LIN {X 0,Y 362.001,Z 141.011,A -85,B 0,C 180,E1 -12973.899,E2 -12973.899} C_VEL
LIN {X 0,Y 361.93,Z 141.028,A -85,B 0,C 180,E1 -12976.934,E2 -12976.934} C_VEL
LIN {X 0,Y 361.889,Z 141.033,A -85,B 0,C 180,E1 -12980.461,E2 -12980.461} C_VEL
LIN {X 0,Y 361.895,Z 141.031,A -85,B 0,C 180,E1 -12984.112,E2 -12984.112} C_VEL
LIN {X 0,Y 361.866,Z 141.033,A -85,B 0,C 180,E1 -12987.782,E2 -12987.782} C_VEL
LIN {X 0,Y 361.849,Z 141.037,A -85,B 0,C 180,E1 -12991.285,E2 -12991.285} C_VEL
LIN {X 0,Y 361.856,Z 141.029,A -85,B 0,C 180,E1 -12994.28,E2 -12994.28} C_VEL
LIN {X 0,Y 361.864,Z 141.03,A -85,B 0,C 180,E1 -12997.223,E2 -12997.223} C_VEL
LIN {X 0,Y 361.836,Z 141.038,A -85,B 0,C 180,E1 -13000.755,E2 -13000.755} C_VEL
LIN {X 0,Y 361.818,Z 141.04,A -85,B 0,C 180,E1 -13004.368,E2 -13004.368} C_VEL
LIN {X 0,Y 361.837,Z 141.036,A -85,B 0,C 180,E1 -13007.568,E2 -13007.568} C_VEL
LIN {X 0,Y 361.871,Z 141.028,A -85,B 0,C 180,E1 -13010.973,E2 -13010.973} C_VEL
LIN {X 0,Y 361.89,Z 141.148,A -85,B 0,C 180,E1 -13012.93,E2 -13012.93} C_VEL
LIN {X 0,Y 365.148,Z 152.964,A -85,B 0,C 180,E1 -13015.855,E2 -13015.855} C_VEL
LIN {X 0,Y 367.944,Z 164.217,A -85,B 0,C 180,E1 -13018.43,E2 -13018.43} C_VEL
LIN {X 0,Y 374.959,Z 180.061,A -85,B 0,C 180,E1 -13019.427,E2 -13019.427} C_VEL
LIN {X 0,Y 380.015,Z 206.73,A -85,B 0,C 180,E1 -13020.441,E2 -13020.441} C_VEL
LIN {X 0,Y 378.027,Z 291.914,A -85,B 0,C 180,E1 -13022.078,E2 -13022.078} C_VEL
LIN {X 0,Y 376.936,Z 331.246,A -85,B 0,C 180,E1 -13022.856,E2 -13022.856} C_VEL
LIN {X 0,Y 375.915,Z 347.066,A -85,B 0,C 180,E1 -13023.377,E2 -13023.377} C_VEL
LIN {X 0,Y 374.628,Z 361.61,A -85,B 0,C 180,E1 -13024.065,E2 -13024.065} C_VEL
LIN {X 0,Y 373.287,Z 375.171,A -85,B 0,C 180,E1 -13024.921,E2 -13024.921} C_VEL
LIN {X 0,Y 371.559,Z 388.868,A -85,B 0,C 180,E1 -13026.004,E2 -13026.004} C_VEL
LIN {X 0,Y 369.85,Z 401.312,A -85,B 0,C 180,E1 -13027.221,E2 -13027.221} C_VEL
LIN {X 0,Y 367.894,Z 413.971,A -85,B 0,C 180,E1 -13028.718,E2 -13028.718} C_VEL
LIN {X 0,Y 366.21,Z 426.144,A -85,B 0,C 180,E1 -13030.483,E2 -13030.483} C_VEL
LIN {X 0,Y 364.434,Z 436.665,A -85,B 0,C 180,E1 -13032.318,E2 -13032.318} C_VEL
LIN {X 0,Y 363.094,Z 445.935,A -85,B 0,C 180,E1 -13034.277,E2 -13034.277} C_VEL
LIN {X 0,Y 361.936,Z 454.664,A -85,B 0,C 180,E1 -13036.525,E2 -13036.525} C_VEL
LIN {X 0,Y 361.134,Z 461.674,A -85,B 0,C 180,E1 -13038.778,E2 -13038.778} C_VEL
LIN {X 0,Y 360.628,Z 467.188,A -85,B 0,C 180,E1 -13041.031,E2 -13041.031} C_VEL
LIN {X 0,Y 360.386,Z 471.36,A -85,B 0,C 180,E1 -13043.28,E2 -13043.28} C_VEL
LIN {X 0,Y 360.3,Z 474.286,A -85,B 0,C 180,E1 -13045.525,E2 -13045.525} C_VEL
LIN {X 0,Y 360.254,Z 476.03,A -85,B 0,C 180,E1 -13047.764,E2 -13047.764} C_VEL
LIN {X 0,Y 360.357,Z 476.63,A -85,B 0,C 180,E1 -13050,E2 -13050} C_VEL
LIN {X 0,Y 360.254,Z 476.023,A -85,B 0,C 180,E1 -13052.236,E2 -13052.236} C_VEL
LIN {X 0,Y 360.302,Z 474.27,A -85,B 0,C 180,E1 -13054.475,E2 -13054.475} C_VEL
LIN {X 0,Y 360.387,Z 471.339,A -85,B 0,C 180,E1 -13056.719,E2 -13056.719} C_VEL
LIN {X 0,Y 360.628,Z 467.166,A -85,B 0,C 180,E1 -13058.969,E2 -13058.969} C_VEL
LIN {X 0,Y 361.126,Z 461.64,A -85,B 0,C 180,E1 -13061.222,E2 -13061.222} C_VEL
LIN {X 0,Y 361.911,Z 454.613,A -85,B 0,C 180,E1 -13063.476,E2 -13063.476} C_VEL
LIN {X 0,Y 363.094,Z 445.876,A -85,B 0,C 180,E1 -13065.723,E2 -13065.723} C_VEL
LIN {X 0,Y 364.405,Z 436.598,A -85,B 0,C 180,E1 -13067.683,E2 -13067.683} C_VEL
LIN {X 0,Y 366.146,Z 426.204,A -85,B 0,C 180,E1 -13069.497,E2 -13069.497} C_VEL
LIN {X 0,Y 367.737,Z 414.949,A -85,B 0,C 180,E1 -13071.145,E2 -13071.145} C_VEL
LIN {X 0,Y 369.626,Z 402.491,A -85,B 0,C 180,E1 -13072.646,E2 -13072.646} C_VEL
LIN {X 0,Y 371.34,Z 390.238,A -85,B 0,C 180,E1 -13073.863,E2 -13073.863} C_VEL
LIN {X 0,Y 373.143,Z 376.327,A -85,B 0,C 180,E1 -13074.981,E2 -13074.981} C_VEL
LIN {X 0,Y 374.607,Z 361.964,A -85,B 0,C 180,E1 -13075.898,E2 -13075.898} C_VEL
LIN {X 0,Y 375.898,Z 346.851,A -85,B 0,C 180,E1 -13076.62,E2 -13076.62} C_VEL
LIN {X 0,Y 376.854,Z 331.928,A -85,B 0,C 180,E1 -13077.113,E2 -13077.113} C_VEL
LIN {X 0,Y 377.84,Z 296.547,A -85,B 0,C 180,E1 -13077.824,E2 -13077.824} C_VEL
LIN {X 0,Y 380.046,Z 207.189,A -85,B 0,C 180,E1 -13079.53,E2 -13079.53} C_VEL
LIN {X 0,Y 375.356,Z 182.22,A -85,B 0,C 180,E1 -13080.473,E2 -13080.473} C_VEL
LIN {X 0,Y 374.41,Z 178.644,A -85,B 0,C 180,E1 -13080.636,E2 -13080.636} C_VEL
LIN {X 0,Y 367.8,Z 163.722,A -85,B 0,C 180,E1 -13081.611,E2 -13081.611} C_VEL
LIN {X 0,Y 364.582,Z 150.743,A -85,B 0,C 180,E1 -13084.657,E2 -13084.657} C_VEL
LIN {X 0,Y 361.877,Z 141.032,A -85,B 0,C 180,E1 -13087.125,E2 -13087.125} C_VEL
LIN {X 0,Y 361.836,Z 141.036,A -85,B 0,C 180,E1 -13090.756,E2 -13090.756} C_VEL
LIN {X 0,Y 361.818,Z 141.037,A -85,B 0,C 180,E1 -13094.369,E2 -13094.369} C_VEL
LIN {X 0,Y 361.837,Z 141.038,A -85,B 0,C 180,E1 -13097.568,E2 -13097.568} C_VEL
LIN {X 0,Y 361.869,Z 141.032,A -85,B 0,C 180,E1 -13100.974,E2 -13100.974} C_VEL
LIN {X 0,Y 361.875,Z 141.026,A -85,B 0,C 180,E1 -13104.655,E2 -13104.655} C_VEL
LIN {X 0,Y 361.838,Z 141.034,A -85,B 0,C 180,E1 -13108.371,E2 -13108.371} C_VEL
LIN {X 0,Y 361.902,Z 141.026,A -85,B 0,C 180,E1 -13110.955,E2 -13110.955} C_VEL
LIN {X 0,Y 361.955,Z 141.02,A -85,B 0,C 180,E1 -13113.475,E2 -13113.475} C_VEL
LIN {X 0,Y 361.88,Z 141.031,A -85,B 0,C 180,E1 -13117.144,E2 -13117.144} C_VEL
LIN {X 0,Y 361.907,Z 141.025,A -85,B 0,C 180,E1 -13120.724,E2 -13120.724} C_VEL
LIN {X 0,Y 361.934,Z 141.021,A -85,B 0,C 180,E1 -13123.066,E2 -13123.066} C_VEL
LIN {X 0,Y 362.001,Z 141.017,A -85,B 0,C 180,E1 -13126.528,E2 -13126.528} C_VEL
LIN {X 0,Y 362.002,Z 141.016,A -85,B 0,C 180,E1 -13129.937,E2 -13129.937} C_VEL
LIN {X 0,Y 362.126,Z 141.001,A -85,B 0,C 180,E1 -13133.313,E2 -13133.313} C_VEL
LIN {X 0,Y 362.279,Z 140.981,A -85,B 0,C 180,E1 -13137.777,E2 -13137.777} C_VEL
LIN {X 0,Y 362.206,Z 140.989,A -85,B 0,C 180,E1 -13141.112,E2 -13141.112} C_VEL
LIN {X 0,Y 362.268,Z 140.986,A -85,B 0,C 180,E1 -13142.224,E2 -13142.224} C_VEL
LIN {X 0,Y 362.126,Z 141.002,A -85,B 0,C 180,E1 -13146.687,E2 -13146.687} C_VEL
LIN {X 0,Y 362.002,Z 141.015,A -85,B 0,C 180,E1 -13150.063,E2 -13150.063} C_VEL
LIN {X 0,Y 361.982,Z 141.015,A -85,B 0,C 180,E1 -13153.887,E2 -13153.887} C_VEL
LIN {X 0,Y 361.912,Z 141.027,A -85,B 0,C 180,E1 -13158.102,E2 -13158.102} C_VEL
LIN {X 0,Y 361.862,Z 141.03,A -85,B 0,C 180,E1 -13161.655,E2 -13161.655} C_VEL
LIN {X 0,Y 361.881,Z 141.016,A -85,B 0,C 180,E1 -13165.294,E2 -13165.294} C_VEL
LIN {X 0,Y 361.857,Z 141.033,A -85,B 0,C 180,E1 -13169.074,E2 -13169.074} C_VEL
LIN {X 0,Y 361.849,Z 141.036,A -85,B 0,C 180,E1 -13172.945,E2 -13172.945} C_VEL
LIN {X 0,Y 361.868,Z 141.035,A -85,B 0,C 180,E1 -13175.637,E2 -13175.637} C_VEL
LIN {X 0,Y 361.826,Z 141.039,A -85,B 0,C 180,E1 -13179.018,E2 -13179.018} C_VEL
LIN {X 0,Y 361.831,Z 141.034,A -85,B 0,C 180,E1 -13182.83,E2 -13182.83} C_VEL
LIN {X 0,Y 361.814,Z 141.04,A -85,B 0,C 180,E1 -13185.948,E2 -13185.948} C_VEL
LIN {X 0,Y 361.812,Z 141.044,A -85,B 0,C 180,E1 -13189.249,E2 -13189.249} C_VEL
LIN {X 0,Y 361.862,Z 141.039,A -85,B 0,C 180,E1 -13192.981,E2 -13192.981} C_VEL
LIN {X 0,Y 361.862,Z 141.096,A -85,B 0,C 180,E1 -13196.481,E2 -13196.481} C_VEL
LIN {X 0,Y 363.496,Z 147.076,A -85,B 0,C 180,E1 -13198.069,E2 -13198.069} C_VEL
LIN {X 0,Y 374.483,Z 169.712,A -85,B 0,C 180,E1 -13199.615,E2 -13199.615} C_VEL
LIN {X 0,Y 380.457,Z 183.537,A -85,B 0,C 180,E1 -13200.441,E2 -13200.441} C_VEL
LIN {X 0,Y 378.69,Z 259.206,A -85,B 0,C 180,E1 -13201.897,E2 -13201.897} C_VEL
LIN {X 0,Y 377.268,Z 311.728,A -85,B 0,C 180,E1 -13202.92,E2 -13202.92} C_VEL
LIN {X 0,Y 376.51,Z 326.715,A -85,B 0,C 180,E1 -13203.411,E2 -13203.411} C_VEL
LIN {X 0,Y 375.568,Z 339.871,A -85,B 0,C 180,E1 -13204.026,E2 -13204.026} C_VEL
LIN {X 0,Y 374.295,Z 353.637,A -85,B 0,C 180,E1 -13204.861,E2 -13204.861} C_VEL
LIN {X 0,Y 372.721,Z 367.614,A -85,B 0,C 180,E1 -13205.936,E2 -13205.936} C_VEL
LIN {X 0,Y 371.026,Z 380.39,A -85,B 0,C 180,E1 -13207.15,E2 -13207.15} C_VEL
LIN {X 0,Y 369.351,Z 392.191,A -85,B 0,C 180,E1 -13208.513,E2 -13208.513} C_VEL
LIN {X 0,Y 367.892,Z 402.228,A -85,B 0,C 180,E1 -13209.888,E2 -13209.888} C_VEL
LIN {X 0,Y 366.261,Z 412.412,A -85,B 0,C 180,E1 -13211.542,E2 -13211.542} C_VEL
LIN {X 0,Y 364.621,Z 422.376,A -85,B 0,C 180,E1 -13213.483,E2 -13213.483} C_VEL
LIN {X 0,Y 363.256,Z 430.637,A -85,B 0,C 180,E1 -13215.433,E2 -13215.433} C_VEL
LIN {X 0,Y 362.559,Z 436.591,A -85,B 0,C 180,E1 -13217.119,E2 -13217.119} C_VEL
LIN {X 0,Y 361.565,Z 443.148,A -85,B 0,C 180,E1 -13219.359,E2 -13219.359} C_VEL
LIN {X 0,Y 361,Z 448.267,A -85,B 0,C 180,E1 -13221.604,E2 -13221.604} C_VEL
LIN {X 0,Y 360.717,Z 451.619,A -85,B 0,C 180,E1 -13223.543,E2 -13223.543} C_VEL
LIN {X 0,Y 360.486,Z 454.105,A -85,B 0,C 180,E1 -13225.527,E2 -13225.527} C_VEL
LIN {X 0,Y 360.345,Z 455.843,A -85,B 0,C 180,E1 -13227.765,E2 -13227.765} C_VEL
LIN {X 0,Y 360.36,Z 456.449,A -85,B 0,C 180,E1 -13230,E2 -13230} C_VEL
LIN {X 0,Y 360.344,Z 455.889,A -85,B 0,C 180,E1 -13232.236,E2 -13232.236} C_VEL
LIN {X 0,Y 360.485,Z 454.211,A -85,B 0,C 180,E1 -13234.473,E2 -13234.473} C_VEL
LIN {X 0,Y 360.743,Z 451.379,A -85,B 0,C 180,E1 -13236.713,E2 -13236.713} C_VEL
LIN {X 0,Y 361.096,Z 447.326,A -85,B 0,C 180,E1 -13238.958,E2 -13238.958} C_VEL
LIN {X 0,Y 361.716,Z 441.948,A -85,B 0,C 180,E1 -13241.204,E2 -13241.204} C_VEL
LIN {X 0,Y 362.788,Z 435.089,A -85,B 0,C 180,E1 -13243.442,E2 -13243.442} C_VEL
LIN {X 0,Y 363.658,Z 428.461,A -85,B 0,C 180,E1 -13245.218,E2 -13245.218} C_VEL
LIN {X 0,Y 363.477,Z 425.34,A -85,B 0,C 180,E1 -13246.009,E2 -13246.009} C_VEL
LIN {X 0,Y 361.593,Z 420.083,A -85,B 0,C 180,E1 -13247.304,E2 -13247.304} C_VEL
LIN {X 0,Y 359.809,Z 414.405,A -85,B 0,C 180,E1 -13248.561,E2 -13248.561} C_VEL
LIN {X 0,Y 359.778,Z 410.579,A -85,B 0,C 180,E1 -13249.281,E2 -13249.281} C_VEL
LIN {X 0,Y 361.534,Z 400.292,A -85,B 0,C 180,E1 -13250.918,E2 -13250.918} C_VEL
LIN {X 0,Y 363.275,Z 388.737,A -85,B 0,C 180,E1 -13252.463,E2 -13252.463} C_VEL
LIN {X 0,Y 365.145,Z 376.221,A -85,B 0,C 180,E1 -13253.841,E2 -13253.841} C_VEL
LIN {X 0,Y 366.799,Z 364.197,A -85,B 0,C 180,E1 -13254.931,E2 -13254.931} C_VEL
LIN {X 0,Y 368.276,Z 350.28,A -85,B 0,C 180,E1 -13255.959,E2 -13255.959} C_VEL
LIN {X 0,Y 369.578,Z 335.892,A -85,B 0,C 180,E1 -13256.779,E2 -13256.779} C_VEL
LIN {X 0,Y 370.58,Z 320.605,A -85,B 0,C 180,E1 -13257.419,E2 -13257.419} C_VEL
LIN {X 0,Y 371.286,Z 305.655,A -85,B 0,C 180,E1 -13257.821,E2 -13257.821} C_VEL
LIN {X 0,Y 374.412,Z 185.887,A -85,B 0,C 180,E1 -13260.146,E2 -13260.146} C_VEL
LIN {X 0,Y 366.261,Z 167.391,A -85,B 0,C 180,E1 -13261.311,E2 -13261.311} C_VEL
LIN {X 0,Y 357.798,Z 150.374,A -85,B 0,C 180,E1 -13262.541,E2 -13262.541} C_VEL
LIN {X 0,Y 356.218,Z 147.141,A -85,B 0,C 180,E1 -13262.8,E2 -13262.8} C_VEL
LIN {X 0,Y 354.822,Z 141.911,A -85,B 0,C 180,E1 -13264.281,E2 -13264.281} C_VEL
LIN {X 0,Y 354.792,Z 141.921,A -85,B 0,C 180,E1 -13267.885,E2 -13267.885} C_VEL
LIN {X 0,Y 354.768,Z 141.921,A -85,B 0,C 180,E1 -13271.168,E2 -13271.168} C_VEL
LIN {X 0,Y 354.759,Z 141.918,A -85,B 0,C 180,E1 -13274.505,E2 -13274.505} C_VEL
LIN {X 0,Y 354.782,Z 141.901,A -85,B 0,C 180,E1 -13277.661,E2 -13277.661} C_VEL
LIN {X 0,Y 354.786,Z 141.915,A -85,B 0,C 180,E1 -13280.662,E2 -13280.662} C_VEL
LIN {X 0,Y 354.819,Z 141.905,A -85,B 0,C 180,E1 -13284.302,E2 -13284.302} C_VEL
LIN {X 0,Y 354.781,Z 141.901,A -85,B 0,C 180,E1 -13287.666,E2 -13287.666} C_VEL
LIN {X 0,Y 354.798,Z 141.913,A -85,B 0,C 180,E1 -13291.614,E2 -13291.614} C_VEL
LIN {X 0,Y 354.806,Z 141.912,A -85,B 0,C 180,E1 -13295.42,E2 -13295.42} C_VEL
LIN {X 0,Y 354.826,Z 141.909,A -85,B 0,C 180,E1 -13299.113,E2 -13299.113} C_VEL
LIN {X 0,Y 354.854,Z 141.906,A -85,B 0,C 180,E1 -13302.718,E2 -13302.718} C_VEL
LIN {X 0,Y 354.952,Z 141.889,A -85,B 0,C 180,E1 -13306.255,E2 -13306.255} C_VEL
LIN {X 0,Y 354.958,Z 141.891,A -85,B 0,C 180,E1 -13309.735,E2 -13309.735} C_VEL
LIN {X 0,Y 355.088,Z 141.878,A -85,B 0,C 180,E1 -13313.18,E2 -13313.18} C_VEL
LIN {X 0,Y 355.229,Z 141.864,A -85,B 0,C 180,E1 -13317.732,E2 -13317.732} C_VEL
LIN {X 0,Y 355.15,Z 141.865,A -85,B 0,C 180,E1 -13321.134,E2 -13321.134} C_VEL
LIN {X 0,Y 355.242,Z 141.859,A -85,B 0,C 180,E1 -13322.268,E2 -13322.268} C_VEL
LIN {X 0,Y 355.092,Z 141.877,A -85,B 0,C 180,E1 -13326.82,E2 -13326.82} C_VEL
LIN {X 0,Y 354.959,Z 141.892,A -85,B 0,C 180,E1 -13330.265,E2 -13330.265} C_VEL
LIN {X 0,Y 354.945,Z 141.89,A -85,B 0,C 180,E1 -13334.019,E2 -13334.019} C_VEL
LIN {X 0,Y 354.892,Z 141.895,A -85,B 0,C 180,E1 -13338.092,E2 -13338.092} C_VEL
LIN {X 0,Y 354.821,Z 141.909,A -85,B 0,C 180,E1 -13341.418,E2 -13341.418} C_VEL
LIN {X 0,Y 354.856,Z 141.91,A -85,B 0,C 180,E1 -13344.576,E2 -13344.576} C_VEL
LIN {X 0,Y 354.811,Z 141.914,A -85,B 0,C 180,E1 -13348.384,E2 -13348.384} C_VEL
LIN {X 0,Y 354.791,Z 141.917,A -85,B 0,C 180,E1 -13352.333,E2 -13352.333} C_VEL
LIN {X 0,Y 354.823,Z 141.911,A -85,B 0,C 180,E1 -13355.699,E2 -13355.699} C_VEL
LIN {X 0,Y 354.825,Z 141.908,A -85,B 0,C 180,E1 -13359.423,E2 -13359.423} C_VEL
LIN {X 0,Y 354.789,Z 141.914,A -85,B 0,C 180,E1 -13362.867,E2 -13362.867} C_VEL
LIN {X 0,Y 354.768,Z 141.921,A -85,B 0,C 180,E1 -13366.103,E2 -13366.103} C_VEL
LIN {X 0,Y 354.789,Z 141.903,A -85,B 0,C 180,E1 -13369.179,E2 -13369.179} C_VEL
LIN {X 0,Y 354.823,Z 141.997,A -85,B 0,C 180,E1 -13372.309,E2 -13372.309} C_VEL
LIN {X 0,Y 358.284,Z 154.417,A -85,B 0,C 180,E1 -13375.473,E2 -13375.473} C_VEL
LIN {X 0,Y 360.699,Z 163.979,A -85,B 0,C 180,E1 -13377.719,E2 -13377.719} C_VEL
LIN {X 0,Y 369.137,Z 182.707,A -85,B 0,C 180,E1 -13378.954,E2 -13378.954} C_VEL
LIN {X 0,Y 373.832,Z 207.936,A -85,B 0,C 180,E1 -13379.932,E2 -13379.932} C_VEL
LIN {X 0,Y 371.72,Z 293.526,A -85,B 0,C 180,E1 -13381.6,E2 -13381.6} C_VEL
LIN {X 0,Y 370.644,Z 331.061,A -85,B 0,C 180,E1 -13382.356,E2 -13382.356} C_VEL
LIN {X 0,Y 369.592,Z 346.876,A -85,B 0,C 180,E1 -13382.885,E2 -13382.885} C_VEL
LIN {X 0,Y 368.24,Z 361.417,A -85,B 0,C 180,E1 -13383.581,E2 -13383.581} C_VEL
LIN {X 0,Y 366.79,Z 375.522,A -85,B 0,C 180,E1 -13384.488,E2 -13384.488} C_VEL
LIN {X 0,Y 365.065,Z 388.673,A -85,B 0,C 180,E1 -13385.549,E2 -13385.549} C_VEL
LIN {X 0,Y 363.264,Z 401.115,A -85,B 0,C 180,E1 -13386.784,E2 -13386.784} C_VEL
LIN {X 0,Y 361.238,Z 413.774,A -85,B 0,C 180,E1 -13388.306,E2 -13388.306} C_VEL
LIN {X 0,Y 359.594,Z 424.506,A -85,B 0,C 180,E1 -13389.87,E2 -13389.87} C_VEL
LIN {X 0,Y 357.901,Z 434.974,A -85,B 0,C 180,E1 -13391.688,E2 -13391.688} C_VEL
LIN {X 0,Y 356.367,Z 444.495,A -85,B 0,C 180,E1 -13393.678,E2 -13393.678} C_VEL
LIN {X 0,Y 355.085,Z 453.175,A -85,B 0,C 180,E1 -13395.89,E2 -13395.89} C_VEL
LIN {X 0,Y 354.319,Z 459.849,A -85,B 0,C 180,E1 -13397.979,E2 -13397.979} C_VEL
LIN {X 0,Y 353.646,Z 465.733,A -85,B 0,C 180,E1 -13400.275,E2 -13400.275} C_VEL
LIN {X 0,Y 353.434,Z 469.236,A -85,B 0,C 180,E1 -13401.999,E2 -13401.999} C_VEL
LIN {X 0,Y 353.24,Z 472.775,A -85,B 0,C 180,E1 -13404.291,E2 -13404.291} C_VEL
LIN {X 0,Y 353.191,Z 475.104,A -85,B 0,C 180,E1 -13406.578,E2 -13406.578} C_VEL
LIN {X 0,Y 353.212,Z 476.276,A -85,B 0,C 180,E1 -13408.86,E2 -13408.86} C_VEL
LIN {X 0,Y 353.212,Z 476.273,A -85,B 0,C 180,E1 -13411.14,E2 -13411.14} C_VEL
LIN {X 0,Y 353.192,Z 475.092,A -85,B 0,C 180,E1 -13413.422,E2 -13413.422} C_VEL
LIN {X 0,Y 353.276,Z 472.5,A -85,B 0,C 180,E1 -13415.908,E2 -13415.908} C_VEL
LIN {X 0,Y 353.483,Z 468.137,A -85,B 0,C 180,E1 -13418.576,E2 -13418.576} C_VEL
LIN {X 0,Y 353.918,Z 462.94,A -85,B 0,C 180,E1 -13420.874,E2 -13420.874} C_VEL
LIN {X 0,Y 354.7,Z 456.298,A -85,B 0,C 180,E1 -13423.171,E2 -13423.171} C_VEL
LIN {X 0,Y 355.816,Z 448.024,A -85,B 0,C 180,E1 -13425.465,E2 -13425.465} C_VEL
LIN {X 0,Y 357.136,Z 439.205,A -85,B 0,C 180,E1 -13427.464,E2 -13427.464} C_VEL
LIN {X 0,Y 358.954,Z 428.612,A -85,B 0,C 180,E1 -13429.442,E2 -13429.442} C_VEL
LIN {X 0,Y 360.619,Z 417.734,A -85,B 0,C 180,E1 -13431.133,E2 -13431.133} C_VEL
LIN {X 0,Y 362.46,Z 405.868,A -85,B 0,C 180,E1 -13432.667,E2 -13432.667} C_VEL
LIN {X 0,Y 364.428,Z 392.897,A -85,B 0,C 180,E1 -13434.041,E2 -13434.041} C_VEL
LIN {X 0,Y 366.257,Z 379.348,A -85,B 0,C 180,E1 -13435.207,E2 -13435.207} C_VEL
LIN {X 0,Y 367.935,Z 364.581,A -85,B 0,C 180,E1 -13436.213,E2 -13436.213} C_VEL
LIN {X 0,Y 369.301,Z 349.62,A -85,B 0,C 180,E1 -13436.985,E2 -13436.985} C_VEL
LIN {X 0,Y 370.334,Z 335.143,A -85,B 0,C 180,E1 -13437.515,E2 -13437.515} C_VEL
LIN {X 0,Y 371.054,Z 317.817,A -85,B 0,C 180,E1 -13437.917,E2 -13437.917} C_VEL
LIN {X 0,Y 373.845,Z 208.655,A -85,B 0,C 180,E1 -13440.033,E2 -13440.033} C_VEL
LIN {X 0,Y 370.11,Z 187.96,A -85,B 0,C 180,E1 -13440.821,E2 -13440.821} C_VEL
LIN {X 0,Y 368.797,Z 181.899,A -85,B 0,C 180,E1 -13441.077,E2 -13441.077} C_VEL
LIN {X 0,Y 361.982,Z 166.85,A -85,B 0,C 180,E1 -13442.067,E2 -13442.067} C_VEL
LIN {X 0,Y 360.565,Z 163.473,A -85,B 0,C 180,E1 -13442.324,E2 -13442.324} C_VEL
LIN {X 0,Y 357.348,Z 150.806,A -85,B 0,C 180,E1 -13445.397,E2 -13445.397} C_VEL
LIN {X 0,Y 354.808,Z 141.912,A -85,B 0,C 180,E1 -13447.74,E2 -13447.74} C_VEL
LIN {X 0,Y 354.789,Z 141.914,A -85,B 0,C 180,E1 -13451.172,E2 -13451.172} C_VEL
LIN {X 0,Y 354.764,Z 141.915,A -85,B 0,C 180,E1 -13454.507,E2 -13454.507} C_VEL
LIN {X 0,Y 354.795,Z 141.916,A -85,B 0,C 180,E1 -13457.663,E2 -13457.663} C_VEL
LIN {X 0,Y 354.816,Z 141.91,A -85,B 0,C 180,E1 -13460.666,E2 -13460.666} C_VEL
LIN {X 0,Y 354.822,Z 141.904,A -85,B 0,C 180,E1 -13464.301,E2 -13464.301} C_VEL
LIN {X 0,Y 354.788,Z 141.913,A -85,B 0,C 180,E1 -13467.667,E2 -13467.667} C_VEL
LIN {X 0,Y 354.87,Z 141.9,A -85,B 0,C 180,E1 -13470.622,E2 -13470.622} C_VEL
LIN {X 0,Y 354.899,Z 141.9,A -85,B 0,C 180,E1 -13474.173,E2 -13474.173} C_VEL
LIN {X 0,Y 354.831,Z 141.91,A -85,B 0,C 180,E1 -13477.894,E2 -13477.894} C_VEL
LIN {X 0,Y 354.924,Z 141.898,A -85,B 0,C 180,E1 -13481.892,E2 -13481.892} C_VEL
LIN {X 0,Y 354.945,Z 141.895,A -85,B 0,C 180,E1 -13485.981,E2 -13485.981} C_VEL
LIN {X 0,Y 354.958,Z 141.893,A -85,B 0,C 180,E1 -13489.735,E2 -13489.735} C_VEL
LIN {X 0,Y 355.091,Z 141.878,A -85,B 0,C 180,E1 -13493.18,E2 -13493.18} C_VEL
LIN {X 0,Y 355.242,Z 141.858,A -85,B 0,C 180,E1 -13497.732,E2 -13497.732} C_VEL
LIN {X 0,Y 355.174,Z 141.865,A -85,B 0,C 180,E1 -13501.134,E2 -13501.134} C_VEL
LIN {X 0,Y 355.23,Z 141.863,A -85,B 0,C 180,E1 -13502.268,E2 -13502.268} C_VEL
LIN {X 0,Y 355.091,Z 141.877,A -85,B 0,C 180,E1 -13506.82,E2 -13506.82} C_VEL
LIN {X 0,Y 354.958,Z 141.895,A -85,B 0,C 180,E1 -13510.265,E2 -13510.265} C_VEL
LIN {X 0,Y 354.925,Z 141.895,A -85,B 0,C 180,E1 -13514.006,E2 -13514.006} C_VEL
LIN {X 0,Y 354.891,Z 141.901,A -85,B 0,C 180,E1 -13518.092,E2 -13518.092} C_VEL
LIN {X 0,Y 354.82,Z 141.906,A -85,B 0,C 180,E1 -13521.418,E2 -13521.418} C_VEL
LIN {X 0,Y 354.849,Z 141.901,A -85,B 0,C 180,E1 -13524.577,E2 -13524.577} C_VEL
LIN {X 0,Y 354.798,Z 141.91,A -85,B 0,C 180,E1 -13528.386,E2 -13528.386} C_VEL
LIN {X 0,Y 354.788,Z 141.915,A -85,B 0,C 180,E1 -13532.333,E2 -13532.333} C_VEL
LIN {X 0,Y 354.822,Z 141.912,A -85,B 0,C 180,E1 -13535.699,E2 -13535.699} C_VEL
LIN {X 0,Y 354.769,Z 141.914,A -85,B 0,C 180,E1 -13539.412,E2 -13539.412} C_VEL
LIN {X 0,Y 354.784,Z 141.912,A -85,B 0,C 180,E1 -13542.866,E2 -13542.866} C_VEL
LIN {X 0,Y 354.763,Z 141.918,A -85,B 0,C 180,E1 -13546.103,E2 -13546.103} C_VEL
LIN {X 0,Y 354.765,Z 141.921,A -85,B 0,C 180,E1 -13549.176,E2 -13549.176} C_VEL
LIN {X 0,Y 354.799,Z 141.914,A -85,B 0,C 180,E1 -13552.405,E2 -13552.405} C_VEL
LIN {X 0,Y 354.837,Z 141.984,A -85,B 0,C 180,E1 -13555.892,E2 -13555.892} C_VEL
LIN {X 0,Y 356.254,Z 147.265,A -85,B 0,C 180,E1 -13557.339,E2 -13557.339} C_VEL
LIN {X 0,Y 366.392,Z 167.617,A -85,B 0,C 180,E1 -13558.817,E2 -13558.817} C_VEL
LIN {X 0,Y 374.282,Z 185.48,A -85,B 0,C 180,E1 -13559.941,E2 -13559.941} C_VEL
LIN {X 0,Y 372.386,Z 261.781,A -85,B 0,C 180,E1 -13561.429,E2 -13561.429} C_VEL
LIN {X 0,Y 370.966,Z 311.944,A -85,B 0,C 180,E1 -13562.421,E2 -13562.421} C_VEL
LIN {X 0,Y 370.176,Z 326.96,A -85,B 0,C 180,E1 -13562.921,E2 -13562.921} C_VEL
LIN {X 0,Y 369.08,Z 342.044,A -85,B 0,C 180,E1 -13563.65,E2 -13563.65} C_VEL
LIN {X 0,Y 367.71,Z 355.821,A -85,B 0,C 180,E1 -13564.53,E2 -13564.53} C_VEL
LIN {X 0,Y 366.05,Z 369.396,A -85,B 0,C 180,E1 -13565.62,E2 -13565.62} C_VEL
LIN {X 0,Y 364.114,Z 383.167,A -85,B 0,C 180,E1 -13566.992,E2 -13566.992} C_VEL
LIN {X 0,Y 362.397,Z 394.521,A -85,B 0,C 180,E1 -13568.379,E2 -13568.379} C_VEL
LIN {X 0,Y 360.568,Z 405.98,A -85,B 0,C 180,E1 -13570.056,E2 -13570.056} C_VEL
LIN {X 0,Y 358.959,Z 415.62,A -85,B 0,C 180,E1 -13571.744,E2 -13571.744} C_VEL
LIN {X 0,Y 357.352,Z 425.066,A -85,B 0,C 180,E1 -13573.725,E2 -13573.725} C_VEL
LIN {X 0,Y 356.073,Z 432.927,A -85,B 0,C 180,E1 -13575.717,E2 -13575.717} C_VEL
LIN {X 0,Y 355.29,Z 438.588,A -85,B 0,C 180,E1 -13577.432,E2 -13577.432} C_VEL
LIN {X 0,Y 354.407,Z 444.758,A -85,B 0,C 180,E1 -13579.719,E2 -13579.719} C_VEL
LIN {X 0,Y 353.855,Z 449.52,A -85,B 0,C 180,E1 -13582.008,E2 -13582.008} C_VEL
LIN {X 0,Y 353.511,Z 453.008,A -85,B 0,C 180,E1 -13584.295,E2 -13584.295} C_VEL
LIN {X 0,Y 353.292,Z 455.315,A -85,B 0,C 180,E1 -13586.579,E2 -13586.579} C_VEL
LIN {X 0,Y 353.25,Z 456.491,A -85,B 0,C 180,E1 -13588.86,E2 -13588.86} C_VEL
LIN {X 0,Y 353.25,Z 456.506,A -85,B 0,C 180,E1 -13591.14,E2 -13591.14} C_VEL
LIN {X 0,Y 353.292,Z 455.39,A -85,B 0,C 180,E1 -13593.421,E2 -13593.421} C_VEL
LIN {X 0,Y 353.51,Z 453.142,A -85,B 0,C 180,E1 -13595.705,E2 -13595.705} C_VEL
LIN {X 0,Y 353.81,Z 449.71,A -85,B 0,C 180,E1 -13597.993,E2 -13597.993} C_VEL
LIN {X 0,Y 354.362,Z 445.009,A -85,B 0,C 180,E1 -13600.282,E2 -13600.282} C_VEL
LIN {X 0,Y 355.271,Z 438.913,A -85,B 0,C 180,E1 -13602.568,E2 -13602.568} C_VEL
LIN {X 0,Y 356.372,Z 431.239,A -85,B 0,C 180,E1 -13604.855,E2 -13604.855} C_VEL
LIN {X 0,Y 357.708,Z 423.051,A -85,B 0,C 180,E1 -13606.846,E2 -13606.846} C_VEL
LIN {X 0,Y 359.404,Z 413.182,A -85,B 0,C 180,E1 -13608.823,E2 -13608.823} C_VEL
LIN {X 0,Y 359.778,Z 410.579,A -85,B 0,C 180,E1 -13609.281,E2 -13609.281} C_VEL
LIN {X 0,Y 359.75,Z 406.674,A -85,B 0,C 180,E1 -13609.989,E2 -13609.989} C_VEL
LIN {X 0,Y 358.058,Z 400.237,A -85,B 0,C 180,E1 -13611.173,E2 -13611.173} C_VEL
LIN {X 0,Y 356.52,Z 393.429,A -85,B 0,C 180,E1 -13612.299,E2 -13612.299} C_VEL
LIN {X 0,Y 356.708,Z 388.903,A -85,B 0,C 180,E1 -13612.904,E2 -13612.904} C_VEL
LIN {X 0,Y 358.638,Z 376.416,A -85,B 0,C 180,E1 -13614.301,E2 -13614.301} C_VEL
LIN {X 0,Y 360.372,Z 364.39,A -85,B 0,C 180,E1 -13615.407,E2 -13615.407} C_VEL
LIN {X 0,Y 361.902,Z 350.472,A -85,B 0,C 180,E1 -13616.452,E2 -13616.452} C_VEL
LIN {X 0,Y 363.278,Z 335.82,A -85,B 0,C 180,E1 -13617.297,E2 -13617.297} C_VEL
LIN {X 0,Y 364.295,Z 320.791,A -85,B 0,C 180,E1 -13617.933,E2 -13617.933} C_VEL
LIN {X 0,Y 365.033,Z 305.833,A -85,B 0,C 180,E1 -13618.341,E2 -13618.341} C_VEL
LIN {X 0,Y 368.243,Z 187.785,A -85,B 0,C 180,E1 -13620.667,E2 -13620.667} C_VEL
LIN {X 0,Y 360.549,Z 170.406,A -85,B 0,C 180,E1 -13621.799,E2 -13621.799} C_VEL
LIN {X 0,Y 352.617,Z 154.371,A -85,B 0,C 180,E1 -13622.988,E2 -13622.988} C_VEL
LIN {X 0,Y 349.021,Z 147.376,A -85,B 0,C 180,E1 -13623.564,E2 -13623.564} C_VEL
LIN {X 0,Y 347.776,Z 142.793,A -85,B 0,C 180,E1 -13624.901,E2 -13624.901} C_VEL
LIN {X 0,Y 347.731,Z 142.794,A -85,B 0,C 180,E1 -13628.796,E2 -13628.796} C_VEL
LIN {X 0,Y 347.741,Z 142.795,A -85,B 0,C 180,E1 -13631.832,E2 -13631.832} C_VEL
LIN {X 0,Y 347.702,Z 142.8,A -85,B 0,C 180,E1 -13635.028,E2 -13635.028} C_VEL
LIN {X 0,Y 347.739,Z 142.782,A -85,B 0,C 180,E1 -13638.4,E2 -13638.4} C_VEL
LIN {X 0,Y 347.763,Z 142.775,A -85,B 0,C 180,E1 -13642.014,E2 -13642.014} C_VEL
LIN {X 0,Y 347.744,Z 142.793,A -85,B 0,C 180,E1 -13645.536,E2 -13645.536} C_VEL
LIN {X 0,Y 347.731,Z 142.772,A -85,B 0,C 180,E1 -13648.299,E2 -13648.299} C_VEL
LIN {X 0,Y 347.745,Z 142.79,A -85,B 0,C 180,E1 -13650.984,E2 -13650.984} C_VEL
LIN {X 0,Y 347.736,Z 142.79,A -85,B 0,C 180,E1 -13653.6,E2 -13653.6} C_VEL
LIN {X 0,Y 347.75,Z 142.795,A -85,B 0,C 180,E1 -13656.159,E2 -13656.159} C_VEL
LIN {X 0,Y 347.779,Z 142.79,A -85,B 0,C 180,E1 -13659.907,E2 -13659.907} C_VEL
LIN {X 0,Y 347.804,Z 142.784,A -85,B 0,C 180,E1 -13663.567,E2 -13663.567} C_VEL
LIN {X 0,Y 347.9,Z 142.767,A -85,B 0,C 180,E1 -13665.971,E2 -13665.971} C_VEL
LIN {X 0,Y 347.899,Z 142.774,A -85,B 0,C 180,E1 -13669.525,E2 -13669.525} C_VEL
LIN {X 0,Y 348.055,Z 142.754,A -85,B 0,C 180,E1 -13673.041,E2 -13673.041} C_VEL
LIN {X 0,Y 348.191,Z 142.74,A -85,B 0,C 180,E1 -13677.686,E2 -13677.686} C_VEL
LIN {X 0,Y 348.121,Z 142.741,A -85,B 0,C 180,E1 -13681.157,E2 -13681.157} C_VEL
LIN {X 0,Y 348.204,Z 142.735,A -85,B 0,C 180,E1 -13682.313,E2 -13682.313} C_VEL
LIN {X 0,Y 348.059,Z 142.754,A -85,B 0,C 180,E1 -13686.958,E2 -13686.958} C_VEL
LIN {X 0,Y 347.899,Z 142.771,A -85,B 0,C 180,E1 -13690.475,E2 -13690.475} C_VEL
LIN {X 0,Y 347.901,Z 142.768,A -85,B 0,C 180,E1 -13694.15,E2 -13694.15} C_VEL
LIN {X 0,Y 347.831,Z 142.774,A -85,B 0,C 180,E1 -13698.259,E2 -13698.259} C_VEL
LIN {X 0,Y 347.771,Z 142.786,A -85,B 0,C 180,E1 -13701.627,E2 -13701.627} C_VEL
LIN {X 0,Y 347.795,Z 142.787,A -85,B 0,C 180,E1 -13705.11,E2 -13705.11} C_VEL
LIN {X 0,Y 347.759,Z 142.792,A -85,B 0,C 180,E1 -13709.014,E2 -13709.014} C_VEL
LIN {X 0,Y 347.744,Z 142.787,A -85,B 0,C 180,E1 -13713.071,E2 -13713.071} C_VEL
LIN {X 0,Y 347.771,Z 142.79,A -85,B 0,C 180,E1 -13716.065,E2 -13716.065} C_VEL
LIN {X 0,Y 347.753,Z 142.792,A -85,B 0,C 180,E1 -13718.792,E2 -13718.792} C_VEL
LIN {X 0,Y 347.752,Z 142.793,A -85,B 0,C 180,E1 -13721.83,E2 -13721.83} C_VEL
LIN {X 0,Y 347.707,Z 142.796,A -85,B 0,C 180,E1 -13725.026,E2 -13725.026} C_VEL
LIN {X 0,Y 347.751,Z 142.789,A -85,B 0,C 180,E1 -13728.397,E2 -13728.397} C_VEL
LIN {X 0,Y 347.749,Z 142.857,A -85,B 0,C 180,E1 -13731.659,E2 -13731.659} C_VEL
LIN {X 0,Y 351.452,Z 155.84,A -85,B 0,C 180,E1 -13735.072,E2 -13735.072} C_VEL
LIN {X 0,Y 353.374,Z 163.554,A -85,B 0,C 180,E1 -13736.961,E2 -13736.961} C_VEL
LIN {X 0,Y 362.998,Z 184.633,A -85,B 0,C 180,E1 -13738.417,E2 -13738.417} C_VEL
LIN {X 0,Y 366.003,Z 199.415,A -85,B 0,C 180,E1 -13739.035,E2 -13739.035} C_VEL
LIN {X 0,Y 367.725,Z 210.403,A -85,B 0,C 180,E1 -13739.439,E2 -13739.439} C_VEL
LIN {X 0,Y 364.484,Z 328.107,A -85,B 0,C 180,E1 -13741.77,E2 -13741.77} C_VEL
LIN {X 0,Y 363.563,Z 343.247,A -85,B 0,C 180,E1 -13742.241,E2 -13742.241} C_VEL
LIN {X 0,Y 362.136,Z 358.705,A -85,B 0,C 180,E1 -13742.944,E2 -13742.944} C_VEL
LIN {X 0,Y 360.665,Z 372.768,A -85,B 0,C 180,E1 -13743.822,E2 -13743.822} C_VEL
LIN {X 0,Y 358.781,Z 386.891,A -85,B 0,C 180,E1 -13744.938,E2 -13744.938} C_VEL
LIN {X 0,Y 356.874,Z 399.623,A -85,B 0,C 180,E1 -13746.189,E2 -13746.189} C_VEL
LIN {X 0,Y 354.775,Z 412.503,A -85,B 0,C 180,E1 -13747.737,E2 -13747.737} C_VEL
LIN {X 0,Y 353.013,Z 423.509,A -85,B 0,C 180,E1 -13749.342,E2 -13749.342} C_VEL
LIN {X 0,Y 351.411,Z 433.284,A -85,B 0,C 180,E1 -13751.035,E2 -13751.035} C_VEL
LIN {X 0,Y 349.883,Z 441.795,A -85,B 0,C 180,E1 -13752.766,E2 -13752.766} C_VEL
LIN {X 0,Y 348.582,Z 450.132,A -85,B 0,C 180,E1 -13754.805,E2 -13754.805} C_VEL
LIN {X 0,Y 347.483,Z 457.969,A -85,B 0,C 180,E1 -13757.145,E2 -13757.145} C_VEL
LIN {X 0,Y 346.699,Z 464.206,A -85,B 0,C 180,E1 -13759.488,E2 -13759.488} C_VEL
LIN {X 0,Y 346.36,Z 469.037,A -85,B 0,C 180,E1 -13761.834,E2 -13761.834} C_VEL
LIN {X 0,Y 346.16,Z 472.576,A -85,B 0,C 180,E1 -13764.174,E2 -13764.174} C_VEL
LIN {X 0,Y 346.114,Z 474.906,A -85,B 0,C 180,E1 -13766.508,E2 -13766.508} C_VEL
LIN {X 0,Y 346.112,Z 476.077,A -85,B 0,C 180,E1 -13768.836,E2 -13768.836} C_VEL
LIN {X 0,Y 346.112,Z 476.075,A -85,B 0,C 180,E1 -13771.163,E2 -13771.163} C_VEL
LIN {X 0,Y 346.115,Z 474.893,A -85,B 0,C 180,E1 -13773.492,E2 -13773.492} C_VEL
LIN {X 0,Y 346.159,Z 472.555,A -85,B 0,C 180,E1 -13775.826,E2 -13775.826} C_VEL
LIN {X 0,Y 346.36,Z 469.013,A -85,B 0,C 180,E1 -13778.166,E2 -13778.166} C_VEL
LIN {X 0,Y 346.697,Z 464.176,A -85,B 0,C 180,E1 -13780.512,E2 -13780.512} C_VEL
LIN {X 0,Y 347.474,Z 457.921,A -85,B 0,C 180,E1 -13782.855,E2 -13782.855} C_VEL
LIN {X 0,Y 348.375,Z 451.262,A -85,B 0,C 180,E1 -13784.875,E2 -13784.875} C_VEL
LIN {X 0,Y 349.692,Z 442.993,A -85,B 0,C 180,E1 -13786.943,E2 -13786.943} C_VEL
LIN {X 0,Y 351.094,Z 434.7,A -85,B 0,C 180,E1 -13788.68,E2 -13788.68} C_VEL
LIN {X 0,Y 352.884,Z 423.785,A -85,B 0,C 180,E1 -13790.602,E2 -13790.602} C_VEL
LIN {X 0,Y 354.768,Z 412.396,A -85,B 0,C 180,E1 -13792.264,E2 -13792.264} C_VEL
LIN {X 0,Y 356.853,Z 399.49,A -85,B 0,C 180,E1 -13793.812,E2 -13793.812} C_VEL
LIN {X 0,Y 358.77,Z 386.714,A -85,B 0,C 180,E1 -13795.063,E2 -13795.063} C_VEL
LIN {X 0,Y 360.634,Z 372.495,A -85,B 0,C 180,E1 -13796.184,E2 -13796.184} C_VEL
LIN {X 0,Y 362.155,Z 358.427,A -85,B 0,C 180,E1 -13797.054,E2 -13797.054} C_VEL
LIN {X 0,Y 363.468,Z 343.768,A -85,B 0,C 180,E1 -13797.728,E2 -13797.728} C_VEL
LIN {X 0,Y 364.439,Z 328.936,A -85,B 0,C 180,E1 -13798.195,E2 -13798.195} C_VEL
LIN {X 0,Y 367.686,Z 209.871,A -85,B 0,C 180,E1 -13800.558,E2 -13800.558} C_VEL
LIN {X 0,Y 364.233,Z 190.385,A -85,B 0,C 180,E1 -13801.315,E2 -13801.315} C_VEL
LIN {X 0,Y 362.802,Z 184.269,A -85,B 0,C 180,E1 -13801.59,E2 -13801.59} C_VEL
LIN {X 0,Y 354.834,Z 166.743,A -85,B 0,C 180,E1 -13802.789,E2 -13802.789} C_VEL
LIN {X 0,Y 353.331,Z 163.371,A -85,B 0,C 180,E1 -13803.04,E2 -13803.04} C_VEL
LIN {X 0,Y 350.399,Z 152.143,A -85,B 0,C 180,E1 -13805.852,E2 -13805.852} C_VEL
LIN {X 0,Y 347.747,Z 142.795,A -85,B 0,C 180,E1 -13808.341,E2 -13808.341} C_VEL
LIN {X 0,Y 347.751,Z 142.795,A -85,B 0,C 180,E1 -13811.83,E2 -13811.83} C_VEL
LIN {X 0,Y 347.706,Z 142.795,A -85,B 0,C 180,E1 -13815.027,E2 -13815.027} C_VEL
LIN {X 0,Y 347.751,Z 142.79,A -85,B 0,C 180,E1 -13818.397,E2 -13818.397} C_VEL
LIN {X 0,Y 347.774,Z 142.786,A -85,B 0,C 180,E1 -13822.012,E2 -13822.012} C_VEL
LIN {X 0,Y 347.745,Z 142.793,A -85,B 0,C 180,E1 -13825.536,E2 -13825.536} C_VEL
LIN {X 0,Y 347.765,Z 142.784,A -85,B 0,C 180,E1 -13829.654,E2 -13829.654} C_VEL
LIN {X 0,Y 347.853,Z 142.776,A -85,B 0,C 180,E1 -13832.745,E2 -13832.745} C_VEL
LIN {X 0,Y 347.786,Z 142.783,A -85,B 0,C 180,E1 -13836.162,E2 -13836.162} C_VEL
LIN {X 0,Y 347.811,Z 142.777,A -85,B 0,C 180,E1 -13839.909,E2 -13839.909} C_VEL
LIN {X 0,Y 347.868,Z 142.778,A -85,B 0,C 180,E1 -13842.359,E2 -13842.359} C_VEL
LIN {X 0,Y 347.899,Z 142.773,A -85,B 0,C 180,E1 -13845.971,E2 -13845.971} C_VEL
LIN {X 0,Y 347.898,Z 142.773,A -85,B 0,C 180,E1 -13849.525,E2 -13849.525} C_VEL
LIN {X 0,Y 348.058,Z 142.755,A -85,B 0,C 180,E1 -13853.042,E2 -13853.042} C_VEL
LIN {X 0,Y 348.204,Z 142.734,A -85,B 0,C 180,E1 -13857.687,E2 -13857.687} C_VEL
LIN {X 0,Y 348.143,Z 142.74,A -85,B 0,C 180,E1 -13861.157,E2 -13861.157} C_VEL
LIN {X 0,Y 348.191,Z 142.74,A -85,B 0,C 180,E1 -13862.314,E2 -13862.314} C_VEL
LIN {X 0,Y 348.057,Z 142.753,A -85,B 0,C 180,E1 -13866.959,E2 -13866.959} C_VEL
LIN {X 0,Y 347.898,Z 142.775,A -85,B 0,C 180,E1 -13870.475,E2 -13870.475} C_VEL
LIN {X 0,Y 347.881,Z 142.774,A -85,B 0,C 180,E1 -13874.137,E2 -13874.137} C_VEL
LIN {X 0,Y 347.831,Z 142.782,A -85,B 0,C 180,E1 -13878.259,E2 -13878.259} C_VEL
LIN {X 0,Y 347.769,Z 142.785,A -85,B 0,C 180,E1 -13881.626,E2 -13881.626} C_VEL
LIN {X 0,Y 347.767,Z 142.776,A -85,B 0,C 180,E1 -13885.112,E2 -13885.112} C_VEL
LIN {X 0,Y 347.745,Z 142.79,A -85,B 0,C 180,E1 -13889.016,E2 -13889.016} C_VEL
LIN {X 0,Y 347.74,Z 142.793,A -85,B 0,C 180,E1 -13891.914,E2 -13891.914} C_VEL
LIN {X 0,Y 347.788,Z 142.786,A -85,B 0,C 180,E1 -13895.875,E2 -13895.875} C_VEL
LIN {X 0,Y 347.732,Z 142.794,A -85,B 0,C 180,E1 -13898.796,E2 -13898.796} C_VEL
LIN {X 0,Y 347.742,Z 142.788,A -85,B 0,C 180,E1 -13901.832,E2 -13901.832} C_VEL
LIN {X 0,Y 347.701,Z 142.796,A -85,B 0,C 180,E1 -13905.028,E2 -13905.028} C_VEL
LIN {X 0,Y 347.74,Z 142.794,A -85,B 0,C 180,E1 -13908.399,E2 -13908.399} C_VEL
LIN {X 0,Y 347.762,Z 142.785,A -85,B 0,C 180,E1 -13912.014,E2 -13912.014} C_VEL
LIN {X 0,Y 347.789,Z 142.898,A -85,B 0,C 180,E1 -13915.277,E2 -13915.277} C_VEL
LIN {X 0,Y 349.099,Z 147.598,A -85,B 0,C 180,E1 -13916.584,E2 -13916.584} C_VEL
LIN {X 0,Y 358.419,Z 165.932,A -85,B 0,C 180,E1 -13917.996,E2 -13917.996} C_VEL
LIN {X 0,Y 367.049,Z 184.914,A -85,B 0,C 180,E1 -13919.267,E2 -13919.267} C_VEL
LIN {X 0,Y 368.151,Z 187.462,A -85,B 0,C 180,E1 -13919.426,E2 -13919.426} C_VEL
LIN {X 0,Y 365.842,Z 275.217,A -85,B 0,C 180,E1 -13921.16,E2 -13921.16} C_VEL
LIN {X 0,Y 364.714,Z 312.16,A -85,B 0,C 180,E1 -13921.907,E2 -13921.907} C_VEL
LIN {X 0,Y 363.88,Z 327.207,A -85,B 0,C 180,E1 -13922.414,E2 -13922.414} C_VEL
LIN {X 0,Y 362.781,Z 341.227,A -85,B 0,C 180,E1 -13923.095,E2 -13923.095} C_VEL
LIN {X 0,Y 361.489,Z 354.048,A -85,B 0,C 180,E1 -13923.904,E2 -13923.904} C_VEL
LIN {X 0,Y 359.793,Z 368.023,A -85,B 0,C 180,E1 -13925.013,E2 -13925.013} C_VEL
LIN {X 0,Y 357.958,Z 380.797,A -85,B 0,C 180,E1 -13926.266,E2 -13926.266} C_VEL
LIN {X 0,Y 356.119,Z 392.598,A -85,B 0,C 180,E1 -13927.673,E2 -13927.673} C_VEL
LIN {X 0,Y 354.554,Z 402.634,A -85,B 0,C 180,E1 -13929.096,E2 -13929.096} C_VEL
LIN {X 0,Y 352.746,Z 412.818,A -85,B 0,C 180,E1 -13930.808,E2 -13930.808} C_VEL
LIN {X 0,Y 350.984,Z 422.779,A -85,B 0,C 180,E1 -13932.821,E2 -13932.821} C_VEL
LIN {X 0,Y 349.377,Z 431.335,A -85,B 0,C 180,E1 -13934.92,E2 -13934.92} C_VEL
LIN {X 0,Y 348.35,Z 438.789,A -85,B 0,C 180,E1 -13937.178,E2 -13937.178} C_VEL
LIN {X 0,Y 347.374,Z 444.96,A -85,B 0,C 180,E1 -13939.509,E2 -13939.509} C_VEL
LIN {X 0,Y 346.792,Z 449.721,A -85,B 0,C 180,E1 -13941.845,E2 -13941.845} C_VEL
LIN {X 0,Y 346.44,Z 453.207,A -85,B 0,C 180,E1 -13944.178,E2 -13944.178} C_VEL
LIN {X 0,Y 346.218,Z 455.513,A -85,B 0,C 180,E1 -13946.509,E2 -13946.509} C_VEL
LIN {X 0,Y 346.152,Z 456.69,A -85,B 0,C 180,E1 -13948.837,E2 -13948.837} C_VEL
LIN {X 0,Y 346.152,Z 456.705,A -85,B 0,C 180,E1 -13951.163,E2 -13951.163} C_VEL
LIN {X 0,Y 346.217,Z 455.588,A -85,B 0,C 180,E1 -13953.491,E2 -13953.491} C_VEL
LIN {X 0,Y 346.439,Z 453.34,A -85,B 0,C 180,E1 -13955.822,E2 -13955.822} C_VEL
LIN {X 0,Y 346.758,Z 449.908,A -85,B 0,C 180,E1 -13958.156,E2 -13958.156} C_VEL
LIN {X 0,Y 347.338,Z 445.208,A -85,B 0,C 180,E1 -13960.492,E2 -13960.492} C_VEL
LIN {X 0,Y 348.331,Z 439.111,A -85,B 0,C 180,E1 -13962.823,E2 -13962.823} C_VEL
LIN {X 0,Y 349.455,Z 431.437,A -85,B 0,C 180,E1 -13965.156,E2 -13965.156} C_VEL
LIN {X 0,Y 350.883,Z 423.248,A -85,B 0,C 180,E1 -13967.184,E2 -13967.184} C_VEL
LIN {X 0,Y 352.634,Z 413.38,A -85,B 0,C 180,E1 -13969.199,E2 -13969.199} C_VEL
LIN {X 0,Y 354.641,Z 402.199,A -85,B 0,C 180,E1 -13971.076,E2 -13971.076} C_VEL
LIN {X 0,Y 356.514,Z 390.101,A -85,B 0,C 180,E1 -13972.76,E2 -13972.76} C_VEL
LIN {X 0,Y 356.708,Z 388.903,A -85,B 0,C 180,E1 -13972.904,E2 -13972.904} C_VEL
LIN {X 0,Y 356.949,Z 384.297,A -85,B 0,C 180,E1 -13973.493,E2 -13973.493} C_VEL
LIN {X 0,Y 355.578,Z 376.762,A -85,B 0,C 180,E1 -13974.503,E2 -13974.503} C_VEL
LIN {X 0,Y 354.067,Z 368.986,A -85,B 0,C 180,E1 -13975.465,E2 -13975.465} C_VEL
LIN {X 0,Y 354.035,Z 363.919,A -85,B 0,C 180,E1 -13975.956,E2 -13975.956} C_VEL
LIN {X 0,Y 355.682,Z 349.612,A -85,B 0,C 180,E1 -13977.031,E2 -13977.031} C_VEL
LIN {X 0,Y 357.104,Z 334.456,A -85,B 0,C 180,E1 -13977.897,E2 -13977.897} C_VEL
LIN {X 0,Y 358.136,Z 320.032,A -85,B 0,C 180,E1 -13978.497,E2 -13978.497} C_VEL
LIN {X 0,Y 358.892,Z 304.454,A -85,B 0,C 180,E1 -13978.911,E2 -13978.911} C_VEL
LIN {X 0,Y 362.103,Z 189.736,A -85,B 0,C 180,E1 -13981.205,E2 -13981.205} C_VEL
LIN {X 0,Y 353.817,Z 171.05,A -85,B 0,C 180,E1 -13982.467,E2 -13982.467} C_VEL
LIN {X 0,Y 345.471,Z 154.707,A -85,B 0,C 180,E1 -13983.758,E2 -13983.758} C_VEL
LIN {X 0,Y 341.791,Z 147.622,A -85,B 0,C 180,E1 -13984.368,E2 -13984.368} C_VEL
LIN {X 0,Y 340.726,Z 143.672,A -85,B 0,C 180,E1 -13985.55,E2 -13985.55} C_VEL
LIN {X 0,Y 340.694,Z 143.676,A -85,B 0,C 180,E1 -13988.382,E2 -13988.382} C_VEL
LIN {X 0,Y 340.691,Z 143.673,A -85,B 0,C 180,E1 -13992.044,E2 -13992.044} C_VEL
LIN {X 0,Y 340.65,Z 143.673,A -85,B 0,C 180,E1 -13996.228,E2 -13996.228} C_VEL
LIN {X 0,Y 340.669,Z 143.664,A -85,B 0,C 180,E1 -13998.688,E2 -13998.688} C_VEL
LIN {X 0,Y 340.719,Z 143.654,A -85,B 0,C 180,E1 -14001.771,E2 -14001.771} C_VEL
LIN {X 0,Y 340.724,Z 143.667,A -85,B 0,C 180,E1 -14005.596,E2 -14005.596} C_VEL
LIN {X 0,Y 340.684,Z 143.648,A -85,B 0,C 180,E1 -14008.954,E2 -14008.954} C_VEL
LIN {X 0,Y 340.691,Z 143.673,A -85,B 0,C 180,E1 -14012.503,E2 -14012.503} C_VEL
LIN {X 0,Y 340.717,Z 143.668,A -85,B 0,C 180,E1 -14015.635,E2 -14015.635} C_VEL
LIN {X 0,Y 340.717,Z 143.667,A -85,B 0,C 180,E1 -14019.472,E2 -14019.472} C_VEL
LIN {X 0,Y 340.763,Z 143.656,A -85,B 0,C 180,E1 -14021.979,E2 -14021.979} C_VEL
LIN {X 0,Y 340.855,Z 143.646,A -85,B 0,C 180,E1 -14025.716,E2 -14025.716} C_VEL
LIN {X 0,Y 340.851,Z 143.651,A -85,B 0,C 180,E1 -14029.305,E2 -14029.305} C_VEL
LIN {X 0,Y 341.002,Z 143.632,A -85,B 0,C 180,E1 -14032.897,E2 -14032.897} C_VEL
LIN {X 0,Y 340.814,Z 143.648,A -85,B 0,C 180,E1 -14035.268,E2 -14035.268} C_VEL
LIN {X 0,Y 341.128,Z 143.62,A -85,B 0,C 180,E1 -14037.638,E2 -14037.638} C_VEL
LIN {X 0,Y 341.092,Z 143.616,A -85,B 0,C 180,E1 -14041.18,E2 -14041.18} C_VEL
LIN {X 0,Y 341.166,Z 143.612,A -85,B 0,C 180,E1 -14042.361,E2 -14042.361} C_VEL
LIN {X 0,Y 341.005,Z 143.634,A -85,B 0,C 180,E1 -14047.103,E2 -14047.103} C_VEL
LIN {X 0,Y 340.851,Z 143.65,A -85,B 0,C 180,E1 -14050.694,E2 -14050.694} C_VEL
LIN {X 0,Y 340.865,Z 143.644,A -85,B 0,C 180,E1 -14054.325,E2 -14054.325} C_VEL
LIN {X 0,Y 340.788,Z 143.652,A -85,B 0,C 180,E1 -14058.44,E2 -14058.44} C_VEL
LIN {X 0,Y 340.719,Z 143.663,A -85,B 0,C 180,E1 -14061.841,E2 -14061.841} C_VEL
LIN {X 0,Y 340.747,Z 143.661,A -85,B 0,C 180,E1 -14065.666,E2 -14065.666} C_VEL
LIN {X 0,Y 340.733,Z 143.666,A -85,B 0,C 180,E1 -14069.671,E2 -14069.671} C_VEL
LIN {X 0,Y 340.696,Z 143.663,A -85,B 0,C 180,E1 -14073.846,E2 -14073.846} C_VEL
LIN {X 0,Y 340.706,Z 143.665,A -85,B 0,C 180,E1 -14076.741,E2 -14076.741} C_VEL
LIN {X 0,Y 340.689,Z 143.668,A -85,B 0,C 180,E1 -14080.247,E2 -14080.247} C_VEL
LIN {X 0,Y 340.653,Z 143.678,A -85,B 0,C 180,E1 -14083.773,E2 -14083.773} C_VEL
LIN {X 0,Y 340.7,Z 143.672,A -85,B 0,C 180,E1 -14087.954,E2 -14087.954} C_VEL
LIN {X 0,Y 340.709,Z 143.73,A -85,B 0,C 180,E1 -14090.985,E2 -14090.985} C_VEL
LIN {X 0,Y 344.232,Z 155.948,A -85,B 0,C 180,E1 -14094.308,E2 -14094.308} C_VEL
LIN {X 0,Y 346.158,Z 163.405,A -85,B 0,C 180,E1 -14096.182,E2 -14096.182} C_VEL
LIN {X 0,Y 355.738,Z 184.078,A -85,B 0,C 180,E1 -14097.687,E2 -14097.687} C_VEL
LIN {X 0,Y 357.738,Z 189.02,A -85,B 0,C 180,E1 -14098.003,E2 -14098.003} C_VEL
LIN {X 0,Y 361.563,Z 210.309,A -85,B 0,C 180,E1 -14098.862,E2 -14098.862} C_VEL
LIN {X 0,Y 359.078,Z 300.399,A -85,B 0,C 180,E1 -14100.666,E2 -14100.666} C_VEL
LIN {X 0,Y 358.128,Z 330.69,A -85,B 0,C 180,E1 -14101.303,E2 -14101.303} C_VEL
LIN {X 0,Y 357.101,Z 345.731,A -85,B 0,C 180,E1 -14101.814,E2 -14101.814} C_VEL
LIN {X 0,Y 355.55,Z 361.032,A -85,B 0,C 180,E1 -14102.561,E2 -14102.561} C_VEL
LIN {X 0,Y 353.944,Z 375.58,A -85,B 0,C 180,E1 -14103.53,E2 -14103.53} C_VEL
LIN {X 0,Y 351.897,Z 389.793,A -85,B 0,C 180,E1 -14104.729,E2 -14104.729} C_VEL
LIN {X 0,Y 349.98,Z 402.017,A -85,B 0,C 180,E1 -14106.006,E2 -14106.006} C_VEL
LIN {X 0,Y 347.785,Z 414.453,A -85,B 0,C 180,E1 -14107.578,E2 -14107.578} C_VEL
LIN {X 0,Y 345.901,Z 425.628,A -85,B 0,C 180,E1 -14109.3,E2 -14109.3} C_VEL
LIN {X 0,Y 344.051,Z 436.071,A -85,B 0,C 180,E1 -14111.232,E2 -14111.232} C_VEL
LIN {X 0,Y 342.402,Z 445.337,A -85,B 0,C 180,E1 -14113.3,E2 -14113.3} C_VEL
LIN {X 0,Y 340.998,Z 454.065,A -85,B 0,C 180,E1 -14115.681,E2 -14115.681} C_VEL
LIN {X 0,Y 340.082,Z 461.076,A -85,B 0,C 180,E1 -14118.073,E2 -14118.073} C_VEL
LIN {X 0,Y 339.432,Z 466.589,A -85,B 0,C 180,E1 -14120.465,E2 -14120.465} C_VEL
LIN {X 0,Y 339.144,Z 470.763,A -85,B 0,C 180,E1 -14122.857,E2 -14122.857} C_VEL
LIN {X 0,Y 339.019,Z 473.689,A -85,B 0,C 180,E1 -14125.243,E2 -14125.243} C_VEL
LIN {X 0,Y 338.987,Z 475.435,A -85,B 0,C 180,E1 -14127.624,E2 -14127.624} C_VEL
LIN {X 0,Y 339.065,Z 476.034,A -85,B 0,C 180,E1 -14130,E2 -14130} C_VEL
LIN {X 0,Y 338.987,Z 475.426,A -85,B 0,C 180,E1 -14132.376,E2 -14132.376} C_VEL
LIN {X 0,Y 339.021,Z 473.671,A -85,B 0,C 180,E1 -14134.756,E2 -14134.756} C_VEL
LIN {X 0,Y 339.144,Z 470.738,A -85,B 0,C 180,E1 -14137.142,E2 -14137.142} C_VEL
LIN {X 0,Y 339.432,Z 466.562,A -85,B 0,C 180,E1 -14139.535,E2 -14139.535} C_VEL
LIN {X 0,Y 340.073,Z 461.035,A -85,B 0,C 180,E1 -14141.927,E2 -14141.927} C_VEL
LIN {X 0,Y 340.912,Z 454.003,A -85,B 0,C 180,E1 -14144.323,E2 -14144.323} C_VEL
LIN {X 0,Y 342.202,Z 446.492,A -85,B 0,C 180,E1 -14146.403,E2 -14146.403} C_VEL
LIN {X 0,Y 343.704,Z 437.437,A -85,B 0,C 180,E1 -14148.478,E2 -14148.478} C_VEL
LIN {X 0,Y 345.667,Z 427.023,A -85,B 0,C 180,E1 -14150.445,E2 -14150.445} C_VEL
LIN {X 0,Y 347.596,Z 415.366,A -85,B 0,C 180,E1 -14152.278,E2 -14152.278} C_VEL
LIN {X 0,Y 349.732,Z 403.106,A -85,B 0,C 180,E1 -14153.855,E2 -14153.855} C_VEL
LIN {X 0,Y 351.885,Z 389.627,A -85,B 0,C 180,E1 -14155.272,E2 -14155.272} C_VEL
LIN {X 0,Y 353.912,Z 375.363,A -85,B 0,C 180,E1 -14156.472,E2 -14156.472} C_VEL
LIN {X 0,Y 355.579,Z 360.775,A -85,B 0,C 180,E1 -14157.437,E2 -14157.437} C_VEL
LIN {X 0,Y 357.041,Z 345.365,A -85,B 0,C 180,E1 -14158.191,E2 -14158.191} C_VEL
LIN {X 0,Y 358.119,Z 330.139,A -85,B 0,C 180,E1 -14158.698,E2 -14158.698} C_VEL
LIN {X 0,Y 361.405,Z 215.271,A -85,B 0,C 180,E1 -14161.02,E2 -14161.02} C_VEL
LIN {X 0,Y 361.439,Z 209.753,A -85,B 0,C 180,E1 -14161.142,E2 -14161.142} C_VEL
LIN {X 0,Y 357.467,Z 188.152,A -85,B 0,C 180,E1 -14162.023,E2 -14162.023} C_VEL
LIN {X 0,Y 351.361,Z 174.464,A -85,B 0,C 180,E1 -14162.968,E2 -14162.968} C_VEL
LIN {X 0,Y 346.042,Z 163.05,A -85,B 0,C 180,E1 -14163.845,E2 -14163.845} C_VEL
LIN {X 0,Y 342.899,Z 151.171,A -85,B 0,C 180,E1 -14166.933,E2 -14166.933} C_VEL
LIN {X 0,Y 340.708,Z 143.669,A -85,B 0,C 180,E1 -14169.015,E2 -14169.015} C_VEL
LIN {X 0,Y 340.676,Z 143.671,A -85,B 0,C 180,E1 -14172.904,E2 -14172.904} C_VEL
LIN {X 0,Y 340.676,Z 143.67,A -85,B 0,C 180,E1 -14177.096,E2 -14177.096} C_VEL
LIN {X 0,Y 340.7,Z 143.669,A -85,B 0,C 180,E1 -14180.248,E2 -14180.248} C_VEL
LIN {X 0,Y 340.711,Z 143.664,A -85,B 0,C 180,E1 -14183.56,E2 -14183.56} C_VEL
LIN {X 0,Y 340.693,Z 143.667,A -85,B 0,C 180,E1 -14186.154,E2 -14186.154} C_VEL
LIN {X 0,Y 340.776,Z 143.654,A -85,B 0,C 180,E1 -14190.333,E2 -14190.333} C_VEL
LIN {X 0,Y 340.806,Z 143.653,A -85,B 0,C 180,E1 -14193.02,E2 -14193.02} C_VEL
LIN {X 0,Y 340.756,Z 143.66,A -85,B 0,C 180,E1 -14195.638,E2 -14195.638} C_VEL
LIN {X 0,Y 340.751,Z 143.658,A -85,B 0,C 180,E1 -14199.475,E2 -14199.475} C_VEL
LIN {X 0,Y 340.859,Z 143.65,A -85,B 0,C 180,E1 -14201.984,E2 -14201.984} C_VEL
LIN {X 0,Y 340.871,Z 143.648,A -85,B 0,C 180,E1 -14205.705,E2 -14205.705} C_VEL
LIN {X 0,Y 340.85,Z 143.652,A -85,B 0,C 180,E1 -14209.306,E2 -14209.306} C_VEL
LIN {X 0,Y 341.005,Z 143.632,A -85,B 0,C 180,E1 -14212.897,E2 -14212.897} C_VEL
LIN {X 0,Y 340.829,Z 143.648,A -85,B 0,C 180,E1 -14215.269,E2 -14215.269} C_VEL
LIN {X 0,Y 341.165,Z 143.611,A -85,B 0,C 180,E1 -14217.639,E2 -14217.639} C_VEL
LIN {X 0,Y 341.111,Z 143.616,A -85,B 0,C 180,E1 -14221.181,E2 -14221.181} C_VEL
LIN {X 0,Y 341.128,Z 143.62,A -85,B 0,C 180,E1 -14222.362,E2 -14222.362} C_VEL
LIN {X 0,Y 340.994,Z 143.63,A -85,B 0,C 180,E1 -14226.469,E2 -14226.469} C_VEL
LIN {X 0,Y 340.883,Z 143.64,A -85,B 0,C 180,E1 -14229.494,E2 -14229.494} C_VEL
LIN {X 0,Y 340.844,Z 143.644,A -85,B 0,C 180,E1 -14233.11,E2 -14233.11} C_VEL
LIN {X 0,Y 340.752,Z 143.657,A -85,B 0,C 180,E1 -14236.783,E2 -14236.783} C_VEL
LIN {X 0,Y 340.764,Z 143.663,A -85,B 0,C 180,E1 -14239.268,E2 -14239.268} C_VEL
LIN {X 0,Y 340.712,Z 143.669,A -85,B 0,C 180,E1 -14243.074,E2 -14243.074} C_VEL
LIN {X 0,Y 340.716,Z 143.645,A -85,B 0,C 180,E1 -14245.669,E2 -14245.669} C_VEL
LIN {X 0,Y 340.706,Z 143.673,A -85,B 0,C 180,E1 -14249.674,E2 -14249.674} C_VEL
LIN {X 0,Y 340.687,Z 143.671,A -85,B 0,C 180,E1 -14252.436,E2 -14252.436} C_VEL
LIN {X 0,Y 340.718,Z 143.666,A -85,B 0,C 180,E1 -14255.279,E2 -14255.279} C_VEL
LIN {X 0,Y 340.694,Z 143.669,A -85,B 0,C 180,E1 -14258.382,E2 -14258.382} C_VEL
LIN {X 0,Y 340.693,Z 143.665,A -85,B 0,C 180,E1 -14262.044,E2 -14262.044} C_VEL
LIN {X 0,Y 340.65,Z 143.676,A -85,B 0,C 180,E1 -14266.227,E2 -14266.227} C_VEL
LIN {X 0,Y 340.67,Z 143.674,A -85,B 0,C 180,E1 -14268.688,E2 -14268.688} C_VEL
LIN {X 0,Y 340.719,Z 143.661,A -85,B 0,C 180,E1 -14271.771,E2 -14271.771} C_VEL
LIN {X 0,Y 340.768,Z 143.822,A -85,B 0,C 180,E1 -14274.636,E2 -14274.636} C_VEL
LIN {X 0,Y 341.905,Z 147.766,A -85,B 0,C 180,E1 -14275.782,E2 -14275.782} C_VEL
LIN {X 0,Y 352.185,Z 167.763,A -85,B 0,C 180,E1 -14277.398,E2 -14277.398} C_VEL
LIN {X 0,Y 360.264,Z 185.46,A -85,B 0,C 180,E1 -14278.63,E2 -14278.63} C_VEL
LIN {X 0,Y 362.019,Z 189.53,A -85,B 0,C 180,E1 -14278.893,E2 -14278.893} C_VEL
LIN {X 0,Y 359.539,Z 277.174,A -85,B 0,C 180,E1 -14280.644,E2 -14280.644} C_VEL
LIN {X 0,Y 358.441,Z 313.542,A -85,B 0,C 180,E1 -14281.41,E2 -14281.41} C_VEL
LIN {X 0,Y 357.57,Z 328.115,A -85,B 0,C 180,E1 -14281.919,E2 -14281.919} C_VEL
LIN {X 0,Y 356.406,Z 342.562,A -85,B 0,C 180,E1 -14282.643,E2 -14282.643} C_VEL
LIN {X 0,Y 354.925,Z 356.233,A -85,B 0,C 180,E1 -14283.543,E2 -14283.543} C_VEL
LIN {X 0,Y 353.17,Z 369.804,A -85,B 0,C 180,E1 -14284.669,E2 -14284.669} C_VEL
LIN {X 0,Y 351.27,Z 382.287,A -85,B 0,C 180,E1 -14285.943,E2 -14285.943} C_VEL
LIN {X 0,Y 349.382,Z 393.864,A -85,B 0,C 180,E1 -14287.374,E2 -14287.374} C_VEL
LIN {X 0,Y 347.904,Z 402.836,A -85,B 0,C 180,E1 -14288.677,E2 -14288.677} C_VEL
LIN {X 0,Y 345.993,Z 413.021,A -85,B 0,C 180,E1 -14290.418,E2 -14290.418} C_VEL
LIN {X 0,Y 344.176,Z 422.981,A -85,B 0,C 180,E1 -14292.471,E2 -14292.471} C_VEL
LIN {X 0,Y 342.426,Z 431.94,A -85,B 0,C 180,E1 -14294.717,E2 -14294.717} C_VEL
LIN {X 0,Y 341.412,Z 438.99,A -85,B 0,C 180,E1 -14296.913,E2 -14296.913} C_VEL
LIN {X 0,Y 340.358,Z 445.161,A -85,B 0,C 180,E1 -14299.29,E2 -14299.29} C_VEL
LIN {X 0,Y 339.756,Z 449.921,A -85,B 0,C 180,E1 -14301.674,E2 -14301.674} C_VEL
LIN {X 0,Y 339.367,Z 453.407,A -85,B 0,C 180,E1 -14304.057,E2 -14304.057} C_VEL
LIN {X 0,Y 339.145,Z 455.712,A -85,B 0,C 180,E1 -14306.436,E2 -14306.436} C_VEL
LIN {X 0,Y 339.054,Z 456.889,A -85,B 0,C 180,E1 -14308.812,E2 -14308.812} C_VEL
LIN {X 0,Y 339.054,Z 456.903,A -85,B 0,C 180,E1 -14311.188,E2 -14311.188} C_VEL
LIN {X 0,Y 339.144,Z 455.786,A -85,B 0,C 180,E1 -14313.564,E2 -14313.564} C_VEL
LIN {X 0,Y 339.365,Z 453.539,A -85,B 0,C 180,E1 -14315.943,E2 -14315.943} C_VEL
LIN {X 0,Y 339.725,Z 450.106,A -85,B 0,C 180,E1 -14318.326,E2 -14318.326} C_VEL
LIN {X 0,Y 340.331,Z 445.406,A -85,B 0,C 180,E1 -14320.711,E2 -14320.711} C_VEL
LIN {X 0,Y 341.391,Z 439.308,A -85,B 0,C 180,E1 -14323.088,E2 -14323.088} C_VEL
LIN {X 0,Y 342.562,Z 431.635,A -85,B 0,C 180,E1 -14325.469,E2 -14325.469} C_VEL
LIN {X 0,Y 344.084,Z 423.446,A -85,B 0,C 180,E1 -14327.534,E2 -14327.534} C_VEL
LIN {X 0,Y 345.908,Z 413.577,A -85,B 0,C 180,E1 -14329.587,E2 -14329.587} C_VEL
LIN {X 0,Y 348.056,Z 401.835,A -85,B 0,C 180,E1 -14331.584,E2 -14331.584} C_VEL
LIN {X 0,Y 350.084,Z 389.636,A -85,B 0,C 180,E1 -14333.291,E2 -14333.291} C_VEL
LIN {X 0,Y 352.165,Z 376.61,A -85,B 0,C 180,E1 -14334.777,E2 -14334.777} C_VEL
LIN {X 0,Y 354.035,Z 363.919,A -85,B 0,C 180,E1 -14335.956,E2 -14335.956} C_VEL
LIN {X 0,Y 354.08,Z 358.745,A -85,B 0,C 180,E1 -14336.423,E2 -14336.423} C_VEL
LIN {X 0,Y 352.531,Z 350.356,A -85,B 0,C 180,E1 -14337.244,E2 -14337.244} C_VEL
LIN {X 0,Y 350.861,Z 341.779,A -85,B 0,C 180,E1 -14337.997,E2 -14337.997} C_VEL
LIN {X 0,Y 350.716,Z 336.315,A -85,B 0,C 180,E1 -14338.353,E2 -14338.353} C_VEL
LIN {X 0,Y 351.847,Z 321.162,A -85,B 0,C 180,E1 -14339.013,E2 -14339.013} C_VEL
LIN {X 0,Y 352.605,Z 306.188,A -85,B 0,C 180,E1 -14339.435,E2 -14339.435} C_VEL
LIN {X 0,Y 355.999,Z 191.628,A -85,B 0,C 180,E1 -14341.762,E2 -14341.762} C_VEL
LIN {X 0,Y 347.581,Z 172.804,A -85,B 0,C 180,E1 -14343.085,E2 -14343.085} C_VEL
LIN {X 0,Y 338.521,Z 155.231,A -85,B 0,C 180,E1 -14344.54,E2 -14344.54} C_VEL
LIN {X 0,Y 334.583,Z 147.822,A -85,B 0,C 180,E1 -14345.226,E2 -14345.226} C_VEL
LIN {X 0,Y 333.683,Z 144.542,A -85,B 0,C 180,E1 -14346.224,E2 -14346.224} C_VEL
LIN {X 0,Y 333.602,Z 144.549,A -85,B 0,C 180,E1 -14349.199,E2 -14349.199} C_VEL
LIN {X 0,Y 333.627,Z 144.551,A -85,B 0,C 180,E1 -14352.499,E2 -14352.499} C_VEL
LIN {X 0,Y 333.595,Z 144.556,A -85,B 0,C 180,E1 -14355.954,E2 -14355.954} C_VEL
LIN {X 0,Y 333.603,Z 144.554,A -85,B 0,C 180,E1 -14359.325,E2 -14359.325} C_VEL
LIN {X 0,Y 333.662,Z 144.529,A -85,B 0,C 180,E1 -14363.169,E2 -14363.169} C_VEL
LIN {X 0,Y 333.674,Z 144.546,A -85,B 0,C 180,E1 -14365.341,E2 -14365.341} C_VEL
LIN {X 0,Y 333.622,Z 144.528,A -85,B 0,C 180,E1 -14368.221,E2 -14368.221} C_VEL
LIN {X 0,Y 333.651,Z 144.545,A -85,B 0,C 180,E1 -14371.022,E2 -14371.022} C_VEL
LIN {X 0,Y 333.665,Z 144.546,A -85,B 0,C 180,E1 -14375.086,E2 -14375.086} C_VEL
LIN {X 0,Y 333.656,Z 144.547,A -85,B 0,C 180,E1 -14379.017,E2 -14379.017} C_VEL
LIN {X 0,Y 333.715,Z 144.534,A -85,B 0,C 180,E1 -14381.585,E2 -14381.585} C_VEL
LIN {X 0,Y 333.809,Z 144.524,A -85,B 0,C 180,E1 -14385.578,E2 -14385.578} C_VEL
LIN {X 0,Y 333.82,Z 144.526,A -85,B 0,C 180,E1 -14389.077,E2 -14389.077} C_VEL
LIN {X 0,Y 333.958,Z 144.51,A -85,B 0,C 180,E1 -14392.746,E2 -14392.746} C_VEL
LIN {X 0,Y 333.78,Z 144.524,A -85,B 0,C 180,E1 -14395.169,E2 -14395.169} C_VEL
LIN {X 0,Y 334.068,Z 144.498,A -85,B 0,C 180,E1 -14397.588,E2 -14397.588} C_VEL
LIN {X 0,Y 334.064,Z 144.492,A -85,B 0,C 180,E1 -14401.205,E2 -14401.205} C_VEL
LIN {X 0,Y 334.102,Z 144.492,A -85,B 0,C 180,E1 -14402.411,E2 -14402.411} C_VEL
LIN {X 0,Y 333.994,Z 144.506,A -85,B 0,C 180,E1 -14406.039,E2 -14406.039} C_VEL
LIN {X 0,Y 333.823,Z 144.521,A -85,B 0,C 180,E1 -14409.696,E2 -14409.696} C_VEL
LIN {X 0,Y 333.799,Z 144.524,A -85,B 0,C 180,E1 -14413.391,E2 -14413.391} C_VEL
LIN {X 0,Y 333.721,Z 144.538,A -85,B 0,C 180,E1 -14417.147,E2 -14417.147} C_VEL
LIN {X 0,Y 333.72,Z 144.543,A -85,B 0,C 180,E1 -14419.691,E2 -14419.691} C_VEL
LIN {X 0,Y 333.672,Z 144.548,A -85,B 0,C 180,E1 -14423.59,E2 -14423.59} C_VEL
LIN {X 0,Y 333.677,Z 144.54,A -85,B 0,C 180,E1 -14426.251,E2 -14426.251} C_VEL
LIN {X 0,Y 333.661,Z 144.549,A -85,B 0,C 180,E1 -14430.366,E2 -14430.366} C_VEL
LIN {X 0,Y 333.64,Z 144.543,A -85,B 0,C 180,E1 -14433.208,E2 -14433.208} C_VEL
LIN {X 0,Y 333.666,Z 144.541,A -85,B 0,C 180,E1 -14436.832,E2 -14436.832} C_VEL
LIN {X 0,Y 333.647,Z 144.549,A -85,B 0,C 180,E1 -14440.767,E2 -14440.767} C_VEL
LIN {X 0,Y 333.594,Z 144.555,A -85,B 0,C 180,E1 -14444.25,E2 -14444.25} C_VEL
LIN {X 0,Y 333.642,Z 144.549,A -85,B 0,C 180,E1 -14447.618,E2 -14447.618} C_VEL
LIN {X 0,Y 333.682,Z 144.56,A -85,B 0,C 180,E1 -14450.267,E2 -14450.267} C_VEL
LIN {X 0,Y 337.523,Z 158.061,A -85,B 0,C 180,E1 -14454.04,E2 -14454.04} C_VEL
LIN {X 0,Y 338.831,Z 163.106,A -85,B 0,C 180,E1 -14455.346,E2 -14455.346} C_VEL
LIN {X 0,Y 348.491,Z 183.422,A -85,B 0,C 180,E1 -14456.92,E2 -14456.92} C_VEL
LIN {X 0,Y 351.938,Z 191.538,A -85,B 0,C 180,E1 -14457.474,E2 -14457.474} C_VEL
LIN {X 0,Y 355.478,Z 211.499,A -85,B 0,C 180,E1 -14458.3,E2 -14458.3} C_VEL
LIN {X 0,Y 352.293,Z 321.637,A -85,B 0,C 180,E1 -14460.536,E2 -14460.536} C_VEL
LIN {X 0,Y 351.486,Z 337.33,A -85,B 0,C 180,E1 -14460.954,E2 -14460.954} C_VEL
LIN {X 0,Y 350.119,Z 353.11,A -85,B 0,C 180,E1 -14461.609,E2 -14461.609} C_VEL
LIN {X 0,Y 348.475,Z 367.683,A -85,B 0,C 180,E1 -14462.45,E2 -14462.45} C_VEL
LIN {X 0,Y 346.661,Z 381.715,A -85,B 0,C 180,E1 -14463.512,E2 -14463.512} C_VEL
LIN {X 0,Y 344.489,Z 395.311,A -85,B 0,C 180,E1 -14464.794,E2 -14464.794} C_VEL
LIN {X 0,Y 342.137,Z 408.886,A -85,B 0,C 180,E1 -14466.387,E2 -14466.387} C_VEL
LIN {X 0,Y 339.977,Z 421.106,A -85,B 0,C 180,E1 -14468.155,E2 -14468.155} C_VEL
LIN {X 0,Y 338.186,Z 431.369,A -85,B 0,C 180,E1 -14469.947,E2 -14469.947} C_VEL
LIN {X 0,Y 336.205,Z 441.397,A -85,B 0,C 180,E1 -14472.041,E2 -14472.041} C_VEL
LIN {X 0,Y 334.721,Z 449.733,A -85,B 0,C 180,E1 -14474.16,E2 -14474.16} C_VEL
LIN {X 0,Y 333.516,Z 457.57,A -85,B 0,C 180,E1 -14476.597,E2 -14476.597} C_VEL
LIN {X 0,Y 332.626,Z 463.807,A -85,B 0,C 180,E1 -14479.038,E2 -14479.038} C_VEL
LIN {X 0,Y 332.222,Z 468.638,A -85,B 0,C 180,E1 -14481.484,E2 -14481.484} C_VEL
LIN {X 0,Y 332.007,Z 472.528,A -85,B 0,C 180,E1 -14484.213,E2 -14484.213} C_VEL
LIN {X 0,Y 331.941,Z 474.509,A -85,B 0,C 180,E1 -14486.358,E2 -14486.358} C_VEL
LIN {X 0,Y 331.919,Z 475.68,A -85,B 0,C 180,E1 -14488.787,E2 -14488.787} C_VEL
LIN {X 0,Y 331.919,Z 475.677,A -85,B 0,C 180,E1 -14491.213,E2 -14491.213} C_VEL
LIN {X 0,Y 331.942,Z 474.495,A -85,B 0,C 180,E1 -14493.642,E2 -14493.642} C_VEL
LIN {X 0,Y 331.993,Z 472.155,A -85,B 0,C 180,E1 -14496.076,E2 -14496.076} C_VEL
LIN {X 0,Y 332.222,Z 468.611,A -85,B 0,C 180,E1 -14498.516,E2 -14498.516} C_VEL
LIN {X 0,Y 332.623,Z 463.773,A -85,B 0,C 180,E1 -14500.962,E2 -14500.962} C_VEL
LIN {X 0,Y 333.493,Z 457.517,A -85,B 0,C 180,E1 -14503.404,E2 -14503.404} C_VEL
LIN {X 0,Y 334.558,Z 450.756,A -85,B 0,C 180,E1 -14505.536,E2 -14505.536} C_VEL
LIN {X 0,Y 335.955,Z 442.586,A -85,B 0,C 180,E1 -14507.658,E2 -14507.658} C_VEL
LIN {X 0,Y 337.537,Z 434.294,A -85,B 0,C 180,E1 -14509.46,E2 -14509.46} C_VEL
LIN {X 0,Y 339.448,Z 423.675,A -85,B 0,C 180,E1 -14511.405,E2 -14511.405} C_VEL
LIN {X 0,Y 341.565,Z 411.989,A -85,B 0,C 180,E1 -14513.173,E2 -14513.173} C_VEL
LIN {X 0,Y 343.819,Z 399.082,A -85,B 0,C 180,E1 -14514.774,E2 -14514.774} C_VEL
LIN {X 0,Y 345.91,Z 386.305,A -85,B 0,C 180,E1 -14516.063,E2 -14516.063} C_VEL
LIN {X 0,Y 347.786,Z 373.188,A -85,B 0,C 180,E1 -14517.14,E2 -14517.14} C_VEL
LIN {X 0,Y 349.405,Z 359.316,A -85,B 0,C 180,E1 -14518.045,E2 -14518.045} C_VEL
LIN {X 0,Y 350.896,Z 344.266,A -85,B 0,C 180,E1 -14518.771,E2 -14518.771} C_VEL
LIN {X 0,Y 351.919,Z 329.926,A -85,B 0,C 180,E1 -14519.252,E2 -14519.252} C_VEL
LIN {X 0,Y 355.325,Z 214.951,A -85,B 0,C 180,E1 -14521.614,E2 -14521.614} C_VEL
LIN {X 0,Y 355.283,Z 210.411,A -85,B 0,C 180,E1 -14521.723,E2 -14521.723} C_VEL
LIN {X 0,Y 351.725,Z 190.877,A -85,B 0,C 180,E1 -14522.54,E2 -14522.54} C_VEL
LIN {X 0,Y 344.011,Z 173.806,A -85,B 0,C 180,E1 -14523.775,E2 -14523.775} C_VEL
LIN {X 0,Y 338.805,Z 162.896,A -85,B 0,C 180,E1 -14524.65,E2 -14524.65} C_VEL
LIN {X 0,Y 335.722,Z 151.618,A -85,B 0,C 180,E1 -14527.693,E2 -14527.693} C_VEL
LIN {X 0,Y 333.654,Z 144.549,A -85,B 0,C 180,E1 -14529.737,E2 -14529.737} C_VEL
LIN {X 0,Y 333.633,Z 144.549,A -85,B 0,C 180,E1 -14532.5,E2 -14532.5} C_VEL
LIN {X 0,Y 333.597,Z 144.555,A -85,B 0,C 180,E1 -14535.955,E2 -14535.955} C_VEL
LIN {X 0,Y 333.648,Z 144.545,A -85,B 0,C 180,E1 -14539.316,E2 -14539.316} C_VEL
LIN {X 0,Y 333.666,Z 144.546,A -85,B 0,C 180,E1 -14543.168,E2 -14543.168} C_VEL
LIN {X 0,Y 333.675,Z 144.544,A -85,B 0,C 180,E1 -14545.342,E2 -14545.342} C_VEL
LIN {X 0,Y 333.704,Z 144.535,A -85,B 0,C 180,E1 -14549.71,E2 -14549.71} C_VEL
LIN {X 0,Y 333.745,Z 144.534,A -85,B 0,C 180,E1 -14552.401,E2 -14552.401} C_VEL
LIN {X 0,Y 333.727,Z 144.541,A -85,B 0,C 180,E1 -14555.091,E2 -14555.091} C_VEL
LIN {X 0,Y 333.685,Z 144.542,A -85,B 0,C 180,E1 -14559.02,E2 -14559.02} C_VEL
LIN {X 0,Y 333.795,Z 144.531,A -85,B 0,C 180,E1 -14561.59,E2 -14561.59} C_VEL
LIN {X 0,Y 333.81,Z 144.528,A -85,B 0,C 180,E1 -14565.577,E2 -14565.577} C_VEL
LIN {X 0,Y 333.82,Z 144.529,A -85,B 0,C 180,E1 -14569.078,E2 -14569.078} C_VEL
LIN {X 0,Y 333.959,Z 144.507,A -85,B 0,C 180,E1 -14572.746,E2 -14572.746} C_VEL
LIN {X 0,Y 333.794,Z 144.525,A -85,B 0,C 180,E1 -14575.169,E2 -14575.169} C_VEL
LIN {X 0,Y 334.102,Z 144.491,A -85,B 0,C 180,E1 -14577.589,E2 -14577.589} C_VEL
LIN {X 0,Y 334.08,Z 144.492,A -85,B 0,C 180,E1 -14581.206,E2 -14581.206} C_VEL
LIN {X 0,Y 333.809,Z 144.527,A -85,B 0,C 180,E1 -14583.621,E2 -14583.621} C_VEL
LIN {X 0,Y 333.964,Z 144.506,A -85,B 0,C 180,E1 -14586.46,E2 -14586.46} C_VEL
LIN {X 0,Y 333.822,Z 144.521,A -85,B 0,C 180,E1 -14589.696,E2 -14589.696} C_VEL
LIN {X 0,Y 333.789,Z 144.523,A -85,B 0,C 180,E1 -14593.392,E2 -14593.392} C_VEL
LIN {X 0,Y 333.702,Z 144.535,A -85,B 0,C 180,E1 -14597.149,E2 -14597.149} C_VEL
LIN {X 0,Y 333.719,Z 144.542,A -85,B 0,C 180,E1 -14599.692,E2 -14599.692} C_VEL
LIN {X 0,Y 333.659,Z 144.548,A -85,B 0,C 180,E1 -14603.591,E2 -14603.591} C_VEL
LIN {X 0,Y 333.652,Z 144.521,A -85,B 0,C 180,E1 -14606.254,E2 -14606.254} C_VEL
LIN {X 0,Y 333.658,Z 144.546,A -85,B 0,C 180,E1 -14610.366,E2 -14610.366} C_VEL
LIN {X 0,Y 333.638,Z 144.552,A -85,B 0,C 180,E1 -14613.208,E2 -14613.208} C_VEL
LIN {X 0,Y 333.676,Z 144.543,A -85,B 0,C 180,E1 -14616.139,E2 -14616.139} C_VEL
LIN {X 0,Y 333.621,Z 144.549,A -85,B 0,C 180,E1 -14619.196,E2 -14619.196} C_VEL
LIN {X 0,Y 333.628,Z 144.545,A -85,B 0,C 180,E1 -14622.499,E2 -14622.499} C_VEL
LIN {X 0,Y 333.594,Z 144.555,A -85,B 0,C 180,E1 -14625.954,E2 -14625.954} C_VEL
LIN {X 0,Y 333.603,Z 144.557,A -85,B 0,C 180,E1 -14629.325,E2 -14629.325} C_VEL
LIN {X 0,Y 333.662,Z 144.55,A -85,B 0,C 180,E1 -14633.169,E2 -14633.169} C_VEL
LIN {X 0,Y 333.719,Z 144.627,A -85,B 0,C 180,E1 -14633.926,E2 -14633.926} C_VEL
LIN {X 0,Y 334.67,Z 148.129,A -85,B 0,C 180,E1 -14634.938,E2 -14634.938} C_VEL
LIN {X 0,Y 345.041,Z 167.682,A -85,B 0,C 180,E1 -14636.628,E2 -14636.628} C_VEL
LIN {X 0,Y 353.431,Z 185.723,A -85,B 0,C 180,E1 -14637.952,E2 -14637.952} C_VEL
LIN {X 0,Y 355.904,Z 191.428,A -85,B 0,C 180,E1 -14638.336,E2 -14638.336} C_VEL
LIN {X 0,Y 353.45,Z 276.103,A -85,B 0,C 180,E1 -14640.058,E2 -14640.058} C_VEL
LIN {X 0,Y 352.288,Z 312.592,A -85,B 0,C 180,E1 -14640.822,E2 -14640.822} C_VEL
LIN {X 0,Y 351.381,Z 327.691,A -85,B 0,C 180,E1 -14641.347,E2 -14641.347} C_VEL
LIN {X 0,Y 350.129,Z 342.319,A -85,B 0,C 180,E1 -14642.081,E2 -14642.081} C_VEL
LIN {X 0,Y 348.59,Z 356.438,A -85,B 0,C 180,E1 -14643.023,E2 -14643.023} C_VEL
LIN {X 0,Y 346.753,Z 370.009,A -85,B 0,C 180,E1 -14644.166,E2 -14644.166} C_VEL
LIN {X 0,Y 344.785,Z 382.491,A -85,B 0,C 180,E1 -14645.461,E2 -14645.461} C_VEL
LIN {X 0,Y 342.801,Z 394.068,A -85,B 0,C 180,E1 -14646.915,E2 -14646.915} C_VEL
LIN {X 0,Y 341.261,Z 403.039,A -85,B 0,C 180,E1 -14648.241,E2 -14648.241} C_VEL
LIN {X 0,Y 339.286,Z 413.223,A -85,B 0,C 180,E1 -14650.014,E2 -14650.014} C_VEL
LIN {X 0,Y 337.377,Z 423.184,A -85,B 0,C 180,E1 -14652.106,E2 -14652.106} C_VEL
LIN {X 0,Y 335.69,Z 431.444,A -85,B 0,C 180,E1 -14654.207,E2 -14654.207} C_VEL
LIN {X 0,Y 334.461,Z 439.192,A -85,B 0,C 180,E1 -14656.636,E2 -14656.636} C_VEL
LIN {X 0,Y 333.36,Z 445.362,A -85,B 0,C 180,E1 -14659.062,E2 -14659.062} C_VEL
LIN {X 0,Y 332.713,Z 450.121,A -85,B 0,C 180,E1 -14661.497,E2 -14661.497} C_VEL
LIN {X 0,Y 332.309,Z 453.606,A -85,B 0,C 180,E1 -14663.93,E2 -14663.93} C_VEL
LIN {X 0,Y 332.074,Z 455.911,A -85,B 0,C 180,E1 -14666.36,E2 -14666.36} C_VEL
LIN {X 0,Y 331.959,Z 457.087,A -85,B 0,C 180,E1 -14668.787,E2 -14668.787} C_VEL
LIN {X 0,Y 331.959,Z 457.102,A -85,B 0,C 180,E1 -14671.213,E2 -14671.213} C_VEL
LIN {X 0,Y 332.073,Z 455.984,A -85,B 0,C 180,E1 -14673.64,E2 -14673.64} C_VEL
LIN {X 0,Y 332.391,Z 453.34,A -85,B 0,C 180,E1 -14676.405,E2 -14676.405} C_VEL
LIN {X 0,Y 332.81,Z 449.251,A -85,B 0,C 180,E1 -14679.113,E2 -14679.113} C_VEL
LIN {X 0,Y 333.525,Z 444.196,A -85,B 0,C 180,E1 -14681.548,E2 -14681.548} C_VEL
LIN {X 0,Y 334.723,Z 437.715,A -85,B 0,C 180,E1 -14683.973,E2 -14683.973} C_VEL
LIN {X 0,Y 335.893,Z 430.725,A -85,B 0,C 180,E1 -14686.095,E2 -14686.095} C_VEL
LIN {X 0,Y 337.526,Z 422.306,A -85,B 0,C 180,E1 -14688.2,E2 -14688.2} C_VEL
LIN {X 0,Y 339.478,Z 412.164,A -85,B 0,C 180,E1 -14690.29,E2 -14690.29} C_VEL
LIN {X 0,Y 341.342,Z 402.589,A -85,B 0,C 180,E1 -14691.939,E2 -14691.939} C_VEL
LIN {X 0,Y 343.437,Z 390.492,A -85,B 0,C 180,E1 -14693.678,E2 -14693.678} C_VEL
LIN {X 0,Y 345.518,Z 378.209,A -85,B 0,C 180,E1 -14695.126,E2 -14695.126} C_VEL
LIN {X 0,Y 347.591,Z 364.629,A -85,B 0,C 180,E1 -14696.426,E2 -14696.426} C_VEL
LIN {X 0,Y 349.374,Z 349.803,A -85,B 0,C 180,E1 -14697.56,E2 -14697.56} C_VEL
LIN {X 0,Y 350.716,Z 336.315,A -85,B 0,C 180,E1 -14698.353,E2 -14698.353} C_VEL
LIN {X 0,Y 350.601,Z 330.761,A -85,B 0,C 180,E1 -14698.684,E2 -14698.684} C_VEL
LIN {X 0,Y 348.75,Z 321.721,A -85,B 0,C 180,E1 -14699.279,E2 -14699.279} C_VEL
LIN {X 0,Y 346.816,Z 312.549,A -85,B 0,C 180,E1 -14699.803,E2 -14699.803} C_VEL
LIN {X 0,Y 346.446,Z 306.791,A -85,B 0,C 180,E1 -14700,E2 -14700} C_VEL
LIN {X 0,Y 349.924,Z 193.604,A -85,B 0,C 180,E1 -14702.336,E2 -14702.336} C_VEL
LIN {X 0,Y 341.636,Z 175.185,A -85,B 0,C 180,E1 -14703.682,E2 -14703.682} C_VEL
LIN {X 0,Y 332.806,Z 158.071,A -85,B 0,C 180,E1 -14705.151,E2 -14705.151} C_VEL
LIN {X 0,Y 327.387,Z 148.139,A -85,B 0,C 180,E1 -14706.099,E2 -14706.099} C_VEL
LIN {X 0,Y 326.608,Z 145.423,A -85,B 0,C 180,E1 -14706.989,E2 -14706.989} C_VEL
LIN {X 0,Y 326.552,Z 145.426,A -85,B 0,C 180,E1 -14710.215,E2 -14710.215} C_VEL
LIN {X 0,Y 326.56,Z 145.433,A -85,B 0,C 180,E1 -14713.526,E2 -14713.526} C_VEL
LIN {X 0,Y 326.573,Z 145.416,A -85,B 0,C 180,E1 -14717.029,E2 -14717.029} C_VEL
LIN {X 0,Y 326.587,Z 145.425,A -85,B 0,C 180,E1 -14720.778,E2 -14720.778} C_VEL
LIN {X 0,Y 326.612,Z 145.419,A -85,B 0,C 180,E1 -14724.48,E2 -14724.48} C_VEL
LIN {X 0,Y 326.605,Z 145.41,A -85,B 0,C 180,E1 -14727.455,E2 -14727.455} C_VEL
LIN {X 0,Y 326.589,Z 145.414,A -85,B 0,C 180,E1 -14730.334,E2 -14730.334} C_VEL
LIN {X 0,Y 326.598,Z 145.423,A -85,B 0,C 180,E1 -14733.135,E2 -14733.135} C_VEL
LIN {X 0,Y 326.593,Z 145.422,A -85,B 0,C 180,E1 -14737.21,E2 -14737.21} C_VEL
LIN {X 0,Y 326.65,Z 145.416,A -85,B 0,C 180,E1 -14741.206,E2 -14741.206} C_VEL
LIN {X 0,Y 326.763,Z 145.403,A -85,B 0,C 180,E1 -14745.435,E2 -14745.435} C_VEL
LIN {X 0,Y 326.761,Z 145.406,A -85,B 0,C 180,E1 -14748.838,E2 -14748.838} C_VEL
LIN {X 0,Y 326.915,Z 145.387,A -85,B 0,C 180,E1 -14752.589,E2 -14752.589} C_VEL
LIN {X 0,Y 326.749,Z 145.4,A -85,B 0,C 180,E1 -14755.064,E2 -14755.064} C_VEL
LIN {X 0,Y 327.012,Z 145.377,A -85,B 0,C 180,E1 -14757.536,E2 -14757.536} C_VEL
LIN {X 0,Y 327.034,Z 145.367,A -85,B 0,C 180,E1 -14761.231,E2 -14761.231} C_VEL
LIN {X 0,Y 327.043,Z 145.371,A -85,B 0,C 180,E1 -14762.463,E2 -14762.463} C_VEL
LIN {X 0,Y 326.947,Z 145.383,A -85,B 0,C 180,E1 -14766.17,E2 -14766.17} C_VEL
LIN {X 0,Y 326.786,Z 145.399,A -85,B 0,C 180,E1 -14769.907,E2 -14769.907} C_VEL
LIN {X 0,Y 326.762,Z 145.4,A -85,B 0,C 180,E1 -14773.685,E2 -14773.685} C_VEL
LIN {X 0,Y 326.666,Z 145.413,A -85,B 0,C 180,E1 -14777.53,E2 -14777.53} C_VEL
LIN {X 0,Y 326.652,Z 145.422,A -85,B 0,C 180,E1 -14780.136,E2 -14780.136} C_VEL
LIN {X 0,Y 326.646,Z 145.422,A -85,B 0,C 180,E1 -14784.129,E2 -14784.129} C_VEL
LIN {X 0,Y 326.629,Z 145.424,A -85,B 0,C 180,E1 -14788.253,E2 -14788.253} C_VEL
LIN {X 0,Y 326.577,Z 145.43,A -85,B 0,C 180,E1 -14791.097,E2 -14791.097} C_VEL
LIN {X 0,Y 326.609,Z 145.418,A -85,B 0,C 180,E1 -14794.019,E2 -14794.019} C_VEL
LIN {X 0,Y 326.628,Z 145.418,A -85,B 0,C 180,E1 -14797.238,E2 -14797.238} C_VEL
LIN {X 0,Y 326.579,Z 145.431,A -85,B 0,C 180,E1 -14801.131,E2 -14801.131} C_VEL
LIN {X 0,Y 326.528,Z 145.433,A -85,B 0,C 180,E1 -14804.743,E2 -14804.743} C_VEL
LIN {X 0,Y 326.577,Z 145.429,A -85,B 0,C 180,E1 -14808.154,E2 -14808.154} C_VEL
LIN {X 0,Y 326.624,Z 145.465,A -85,B 0,C 180,E1 -14809.527,E2 -14809.527} C_VEL
LIN {X 0,Y 330.18,Z 157.818,A -85,B 0,C 180,E1 -14813.11,E2 -14813.11} C_VEL
LIN {X 0,Y 331.571,Z 162.787,A -85,B 0,C 180,E1 -14814.472,E2 -14814.472} C_VEL
LIN {X 0,Y 341.364,Z 183.065,A -85,B 0,C 180,E1 -14816.134,E2 -14816.134} C_VEL
LIN {X 0,Y 346.196,Z 194.14,A -85,B 0,C 180,E1 -14816.934,E2 -14816.934} C_VEL
LIN {X 0,Y 349.434,Z 212.607,A -85,B 0,C 180,E1 -14817.716,E2 -14817.716} C_VEL
LIN {X 0,Y 345.956,Z 326.058,A -85,B 0,C 180,E1 -14820.067,E2 -14820.067} C_VEL
LIN {X 0,Y 344.906,Z 341.765,A -85,B 0,C 180,E1 -14820.555,E2 -14820.555} C_VEL
LIN {X 0,Y 343.423,Z 356.828,A -85,B 0,C 180,E1 -14821.254,E2 -14821.254} C_VEL
LIN {X 0,Y 341.674,Z 371.492,A -85,B 0,C 180,E1 -14822.187,E2 -14822.187} C_VEL
LIN {X 0,Y 339.768,Z 384.721,A -85,B 0,C 180,E1 -14823.263,E2 -14823.263} C_VEL
LIN {X 0,Y 337.588,Z 397.738,A -85,B 0,C 180,E1 -14824.572,E2 -14824.572} C_VEL
LIN {X 0,Y 335.382,Z 409.763,A -85,B 0,C 180,E1 -14826.046,E2 -14826.046} C_VEL
LIN {X 0,Y 333.334,Z 420.908,A -85,B 0,C 180,E1 -14827.696,E2 -14827.696} C_VEL
LIN {X 0,Y 331.466,Z 431.171,A -85,B 0,C 180,E1 -14829.522,E2 -14829.522} C_VEL
LIN {X 0,Y 329.362,Z 441.197,A -85,B 0,C 180,E1 -14831.655,E2 -14831.655} C_VEL
LIN {X 0,Y 327.82,Z 449.533,A -85,B 0,C 180,E1 -14833.817,E2 -14833.817} C_VEL
LIN {X 0,Y 326.546,Z 457.371,A -85,B 0,C 180,E1 -14836.305,E2 -14836.305} C_VEL
LIN {X 0,Y 325.601,Z 463.608,A -85,B 0,C 180,E1 -14838.798,E2 -14838.798} C_VEL
LIN {X 0,Y 325.139,Z 468.439,A -85,B 0,C 180,E1 -14841.297,E2 -14841.297} C_VEL
LIN {X 0,Y 324.923,Z 472.52,A -85,B 0,C 180,E1 -14844.248,E2 -14844.248} C_VEL
LIN {X 0,Y 324.847,Z 474.31,A -85,B 0,C 180,E1 -14846.279,E2 -14846.279} C_VEL
LIN {X 0,Y 324.827,Z 475.481,A -85,B 0,C 180,E1 -14848.76,E2 -14848.76} C_VEL
LIN {X 0,Y 324.827,Z 475.478,A -85,B 0,C 180,E1 -14851.24,E2 -14851.24} C_VEL
LIN {X 0,Y 324.848,Z 474.295,A -85,B 0,C 180,E1 -14853.721,E2 -14853.721} C_VEL
LIN {X 0,Y 324.893,Z 471.955,A -85,B 0,C 180,E1 -14856.209,E2 -14856.209} C_VEL
LIN {X 0,Y 325.139,Z 468.41,A -85,B 0,C 180,E1 -14858.703,E2 -14858.703} C_VEL
LIN {X 0,Y 325.597,Z 463.571,A -85,B 0,C 180,E1 -14861.202,E2 -14861.202} C_VEL
LIN {X 0,Y 326.521,Z 457.315,A -85,B 0,C 180,E1 -14863.696,E2 -14863.696} C_VEL
LIN {X 0,Y 327.82,Z 449.462,A -85,B 0,C 180,E1 -14866.183,E2 -14866.183} C_VEL
LIN {X 0,Y 329.337,Z 441.116,A -85,B 0,C 180,E1 -14868.347,E2 -14868.347} C_VEL
LIN {X 0,Y 331.433,Z 431.073,A -85,B 0,C 180,E1 -14870.48,E2 -14870.48} C_VEL
LIN {X 0,Y 333.331,Z 420.8,A -85,B 0,C 180,E1 -14872.304,E2 -14872.304} C_VEL
LIN {X 0,Y 335.606,Z 408.563,A -85,B 0,C 180,E1 -14874.101,E2 -14874.101} C_VEL
LIN {X 0,Y 338.06,Z 394.943,A -85,B 0,C 180,E1 -14875.72,E2 -14875.72} C_VEL
LIN {X 0,Y 340.285,Z 381.29,A -85,B 0,C 180,E1 -14877.025,E2 -14877.025} C_VEL
LIN {X 0,Y 342.204,Z 367.401,A -85,B 0,C 180,E1 -14878.085,E2 -14878.085} C_VEL
LIN {X 0,Y 343.899,Z 352.583,A -85,B 0,C 180,E1 -14878.953,E2 -14878.953} C_VEL
LIN {X 0,Y 345.182,Z 337.632,A -85,B 0,C 180,E1 -14879.587,E2 -14879.587} C_VEL
LIN {X 0,Y 346.068,Z 322.258,A -85,B 0,C 180,E1 -14880.006,E2 -14880.006} C_VEL
LIN {X 0,Y 349.321,Z 212.092,A -85,B 0,C 180,E1 -14882.285,E2 -14882.285} C_VEL
LIN {X 0,Y 345.943,Z 193.508,A -85,B 0,C 180,E1 -14883.085,E2 -14883.085} C_VEL
LIN {X 0,Y 337.537,Z 174.92,A -85,B 0,C 180,E1 -14884.479,E2 -14884.479} C_VEL
LIN {X 0,Y 331.49,Z 162.554,A -85,B 0,C 180,E1 -14885.552,E2 -14885.552} C_VEL
LIN {X 0,Y 328.313,Z 151.367,A -85,B 0,C 180,E1 -14888.699,E2 -14888.699} C_VEL
LIN {X 0,Y 326.603,Z 145.426,A -85,B 0,C 180,E1 -14890.476,E2 -14890.476} C_VEL
LIN {X 0,Y 326.562,Z 145.433,A -85,B 0,C 180,E1 -14893.526,E2 -14893.526} C_VEL
LIN {X 0,Y 326.576,Z 145.426,A -85,B 0,C 180,E1 -14897.028,E2 -14897.028} C_VEL
LIN {X 0,Y 326.612,Z 145.424,A -85,B 0,C 180,E1 -14900.773,E2 -14900.773} C_VEL
LIN {X 0,Y 326.613,Z 145.418,A -85,B 0,C 180,E1 -14904.481,E2 -14904.481} C_VEL
LIN {X 0,Y 326.609,Z 145.42,A -85,B 0,C 180,E1 -14907.456,E2 -14907.456} C_VEL
LIN {X 0,Y 326.662,Z 145.412,A -85,B 0,C 180,E1 -14910.341,E2 -14910.341} C_VEL
LIN {X 0,Y 326.691,Z 145.415,A -85,B 0,C 180,E1 -14914.517,E2 -14914.517} C_VEL
LIN {X 0,Y 326.649,Z 145.422,A -85,B 0,C 180,E1 -14918.546,E2 -14918.546} C_VEL
LIN {X 0,Y 326.746,Z 145.409,A -85,B 0,C 180,E1 -14921.178,E2 -14921.178} C_VEL
LIN {X 0,Y 326.765,Z 145.407,A -85,B 0,C 180,E1 -14925.433,E2 -14925.433} C_VEL
LIN {X 0,Y 326.76,Z 145.406,A -85,B 0,C 180,E1 -14928.839,E2 -14928.839} C_VEL
LIN {X 0,Y 326.916,Z 145.383,A -85,B 0,C 180,E1 -14932.589,E2 -14932.589} C_VEL
LIN {X 0,Y 326.762,Z 145.401,A -85,B 0,C 180,E1 -14935.065,E2 -14935.065} C_VEL
LIN {X 0,Y 327.043,Z 145.37,A -85,B 0,C 180,E1 -14937.537,E2 -14937.537} C_VEL
LIN {X 0,Y 327.048,Z 145.368,A -85,B 0,C 180,E1 -14941.231,E2 -14941.231} C_VEL
LIN {X 0,Y 326.757,Z 145.405,A -85,B 0,C 180,E1 -14943.7,E2 -14943.7} C_VEL
LIN {X 0,Y 326.926,Z 145.384,A -85,B 0,C 180,E1 -14946.448,E2 -14946.448} C_VEL
LIN {X 0,Y 326.785,Z 145.399,A -85,B 0,C 180,E1 -14949.907,E2 -14949.907} C_VEL
LIN {X 0,Y 326.745,Z 145.401,A -85,B 0,C 180,E1 -14953.686,E2 -14953.686} C_VEL
LIN {X 0,Y 326.653,Z 145.413,A -85,B 0,C 180,E1 -14957.531,E2 -14957.531} C_VEL
LIN {X 0,Y 326.649,Z 145.417,A -85,B 0,C 180,E1 -14960.136,E2 -14960.136} C_VEL
LIN {X 0,Y 326.632,Z 145.417,A -85,B 0,C 180,E1 -14964.131,E2 -14964.131} C_VEL
LIN {X 0,Y 326.6,Z 145.413,A -85,B 0,C 180,E1 -14968.083,E2 -14968.083} C_VEL
LIN {X 0,Y 326.574,Z 145.427,A -85,B 0,C 180,E1 -14971.097,E2 -14971.097} C_VEL
LIN {X 0,Y 326.608,Z 145.42,A -85,B 0,C 180,E1 -14974.019,E2 -14974.019} C_VEL
LIN {X 0,Y 326.624,Z 145.419,A -85,B 0,C 180,E1 -14977.237,E2 -14977.237} C_VEL
LIN {X 0,Y 326.545,Z 145.434,A -85,B 0,C 180,E1 -14981.124,E2 -14981.124} C_VEL
LIN {X 0,Y 326.56,Z 145.431,A -85,B 0,C 180,E1 -14983.526,E2 -14983.526} C_VEL
LIN {X 0,Y 326.573,Z 145.429,A -85,B 0,C 180,E1 -14987.029,E2 -14987.029} C_VEL
LIN {X 0,Y 326.572,Z 145.423,A -85,B 0,C 180,E1 -14990.782,E2 -14990.782} C_VEL
LIN {X 0,Y 326.643,Z 145.527,A -85,B 0,C 180,E1 -14993.201,E2 -14993.201} C_VEL
LIN {X 0,Y 327.409,Z 148.23,A -85,B 0,C 180,E1 -14994.037,E2 -14994.037} C_VEL
LIN {X 0,Y 337.022,Z 166.089,A -85,B 0,C 180,E1 -14995.677,E2 -14995.677} C_VEL
LIN {X 0,Y 344.603,Z 181.561,A -85,B 0,C 180,E1 -14996.919,E2 -14996.919} C_VEL
LIN {X 0,Y 349.825,Z 193.557,A -85,B 0,C 180,E1 -14997.765,E2 -14997.765} C_VEL
LIN {X 0,Y 347.364,Z 275.165,A -85,B 0,C 180,E1 -14999.45,E2 -14999.45} C_VEL
LIN {X 0,Y 346.109,Z 312.808,A -85,B 0,C 180,E1 -15000.25,E2 -15000.25} C_VEL
LIN {X 0,Y 345.169,Z 327.938,A -85,B 0,C 180,E1 -15000.784,E2 -15000.784} C_VEL
LIN {X 0,Y 343.84,Z 342.968,A -85,B 0,C 180,E1 -15001.554,E2 -15001.554} C_VEL
LIN {X 0,Y 342.288,Z 356.644,A -85,B 0,C 180,E1 -15002.485,E2 -15002.485} C_VEL
LIN {X 0,Y 340.381,Z 370.213,A -85,B 0,C 180,E1 -15003.646,E2 -15003.646} C_VEL
LIN {X 0,Y 338.331,Z 382.694,A -85,B 0,C 180,E1 -15004.961,E2 -15004.961} C_VEL
LIN {X 0,Y 336.254,Z 394.271,A -85,B 0,C 180,E1 -15006.439,E2 -15006.439} C_VEL
LIN {X 0,Y 334.629,Z 403.243,A -85,B 0,C 180,E1 -15007.787,E2 -15007.787} C_VEL
LIN {X 0,Y 332.584,Z 413.426,A -85,B 0,C 180,E1 -15009.594,E2 -15009.594} C_VEL
LIN {X 0,Y 330.591,Z 423.386,A -85,B 0,C 180,E1 -15011.726,E2 -15011.726} C_VEL
LIN {X 0,Y 328.836,Z 431.646,A -85,B 0,C 180,E1 -15013.869,E2 -15013.869} C_VEL
LIN {X 0,Y 327.508,Z 439.393,A -85,B 0,C 180,E1 -15016.347,E2 -15016.347} C_VEL
LIN {X 0,Y 326.368,Z 445.562,A -85,B 0,C 180,E1 -15018.825,E2 -15018.825} C_VEL
LIN {X 0,Y 325.669,Z 450.321,A -85,B 0,C 180,E1 -15021.312,E2 -15021.312} C_VEL
LIN {X 0,Y 325.24,Z 453.806,A -85,B 0,C 180,E1 -15023.798,E2 -15023.798} C_VEL
LIN {X 0,Y 325.005,Z 456.109,A -85,B 0,C 180,E1 -15026.28,E2 -15026.28} C_VEL
LIN {X 0,Y 324.867,Z 457.286,A -85,B 0,C 180,E1 -15028.76,E2 -15028.76} C_VEL
LIN {X 0,Y 324.867,Z 457.301,A -85,B 0,C 180,E1 -15031.24,E2 -15031.24} C_VEL
LIN {X 0,Y 325.004,Z 456.182,A -85,B 0,C 180,E1 -15033.72,E2 -15033.72} C_VEL
LIN {X 0,Y 325.272,Z 453.788,A -85,B 0,C 180,E1 -15036.33,E2 -15036.33} C_VEL
LIN {X 0,Y 325.638,Z 450.503,A -85,B 0,C 180,E1 -15038.689,E2 -15038.689} C_VEL
LIN {X 0,Y 326.341,Z 445.802,A -85,B 0,C 180,E1 -15041.176,E2 -15041.176} C_VEL
LIN {X 0,Y 327.483,Z 439.706,A -85,B 0,C 180,E1 -15043.655,E2 -15043.655} C_VEL
LIN {X 0,Y 328.828,Z 432.031,A -85,B 0,C 180,E1 -15046.132,E2 -15046.132} C_VEL
LIN {X 0,Y 330.493,Z 423.841,A -85,B 0,C 180,E1 -15048.28,E2 -15048.28} C_VEL
LIN {X 0,Y 332.511,Z 413.971,A -85,B 0,C 180,E1 -15050.411,E2 -15050.411} C_VEL
LIN {X 0,Y 334.726,Z 402.738,A -85,B 0,C 180,E1 -15052.404,E2 -15052.404} C_VEL
LIN {X 0,Y 336.945,Z 390.686,A -85,B 0,C 180,E1 -15054.163,E2 -15054.163} C_VEL
LIN {X 0,Y 339.091,Z 378.404,A -85,B 0,C 180,E1 -15055.636,E2 -15055.636} C_VEL
LIN {X 0,Y 341.22,Z 364.971,A -85,B 0,C 180,E1 -15056.945,E2 -15056.945} C_VEL
LIN {X 0,Y 342.98,Z 351.048,A -85,B 0,C 180,E1 -15058.035,E2 -15058.035} C_VEL
LIN {X 0,Y 344.463,Z 336.731,A -85,B 0,C 180,E1 -15058.902,E2 -15058.902} C_VEL
LIN {X 0,Y 345.659,Z 321.348,A -85,B 0,C 180,E1 -15059.584,E2 -15059.584} C_VEL
LIN {X 0,Y 346.446,Z 306.791,A -85,B 0,C 180,E1 -15060,E2 -15060} C_VEL
LIN {X 0,Y 346.073,Z 301.006,A -85,B 0,C 180,E1 -15060.19,E2 -15060.19} C_VEL
LIN {X 0,Y 341.673,Z 282.386,A -85,B 0,C 180,E1 -15061.063,E2 -15061.063} C_VEL
LIN {X 0,Y 341.296,Z 276.585,A -85,B 0,C 180,E1 -15061.238,E2 -15061.238} C_VEL
LIN {X 0,Y 343.882,Z 195.646,A -85,B 0,C 180,E1 -15062.931,E2 -15062.931} C_VEL
LIN {X 0,Y 335.551,Z 177.2,A -85,B 0,C 180,E1 -15064.331,E2 -15064.331} C_VEL
LIN {X 0,Y 326.934,Z 160.481,A -85,B 0,C 180,E1 -15065.819,E2 -15065.819} C_VEL
LIN {X 0,Y 320.124,Z 148.276,A -85,B 0,C 180,E1 -15067.083,E2 -15067.083} C_VEL
LIN {X 0,Y 319.55,Z 146.309,A -85,B 0,C 180,E1 -15067.777,E2 -15067.777} C_VEL
LIN {X 0,Y 319.504,Z 146.314,A -85,B 0,C 180,E1 -15071.592,E2 -15071.592} C_VEL
LIN {X 0,Y 319.487,Z 146.312,A -85,B 0,C 180,E1 -15074.743,E2 -15074.743} C_VEL
LIN {X 0,Y 319.551,Z 146.29,A -85,B 0,C 180,E1 -15077.016,E2 -15077.016} C_VEL
LIN {X 0,Y 319.546,Z 146.307,A -85,B 0,C 180,E1 -15080.371,E2 -15080.371} C_VEL
LIN {X 0,Y 319.579,Z 146.295,A -85,B 0,C 180,E1 -15084.458,E2 -15084.458} C_VEL
LIN {X 0,Y 319.521,Z 146.284,A -85,B 0,C 180,E1 -15088.137,E2 -15088.137} C_VEL
LIN {X 0,Y 319.57,Z 146.301,A -85,B 0,C 180,E1 -15091.605,E2 -15091.605} C_VEL
LIN {X 0,Y 319.542,Z 146.305,A -85,B 0,C 180,E1 -15095.299,E2 -15095.299} C_VEL
LIN {X 0,Y 319.565,Z 146.296,A -85,B 0,C 180,E1 -15098.045,E2 -15098.045} C_VEL
LIN {X 0,Y 319.59,Z 146.293,A -85,B 0,C 180,E1 -15102.069,E2 -15102.069} C_VEL
LIN {X 0,Y 319.732,Z 146.274,A -85,B 0,C 180,E1 -15106.008,E2 -15106.008} C_VEL
LIN {X 0,Y 319.738,Z 146.275,A -85,B 0,C 180,E1 -15109.872,E2 -15109.872} C_VEL
LIN {X 0,Y 319.9,Z 146.262,A -85,B 0,C 180,E1 -15113.693,E2 -15113.693} C_VEL
LIN {X 0,Y 319.958,Z 146.255,A -85,B 0,C 180,E1 -15117.482,E2 -15117.482} C_VEL
LIN {X 0,Y 320.004,Z 146.243,A -85,B 0,C 180,E1 -15121.258,E2 -15121.258} C_VEL
LIN {X 0,Y 319.729,Z 146.276,A -85,B 0,C 180,E1 -15123.781,E2 -15123.781} C_VEL
LIN {X 0,Y 319.904,Z 146.26,A -85,B 0,C 180,E1 -15126.306,E2 -15126.306} C_VEL
LIN {X 0,Y 319.738,Z 146.278,A -85,B 0,C 180,E1 -15130.128,E2 -15130.128} C_VEL
LIN {X 0,Y 319.734,Z 146.275,A -85,B 0,C 180,E1 -15133.992,E2 -15133.992} C_VEL
LIN {X 0,Y 319.626,Z 146.288,A -85,B 0,C 180,E1 -15137.929,E2 -15137.929} C_VEL
LIN {X 0,Y 319.6,Z 146.303,A -85,B 0,C 180,E1 -15140.6,E2 -15140.6} C_VEL
LIN {X 0,Y 319.586,Z 146.305,A -85,B 0,C 180,E1 -15144.697,E2 -15144.697} C_VEL
LIN {X 0,Y 319.559,Z 146.305,A -85,B 0,C 180,E1 -15148.936,E2 -15148.936} C_VEL
LIN {X 0,Y 319.527,Z 146.308,A -85,B 0,C 180,E1 -15151.862,E2 -15151.862} C_VEL
LIN {X 0,Y 319.581,Z 146.301,A -85,B 0,C 180,E1 -15155.543,E2 -15155.543} C_VEL
LIN {X 0,Y 319.558,Z 146.302,A -85,B 0,C 180,E1 -15158.01,E2 -15158.01} C_VEL
LIN {X 0,Y 319.527,Z 146.309,A -85,B 0,C 180,E1 -15161.597,E2 -15161.597} C_VEL
LIN {X 0,Y 319.489,Z 146.311,A -85,B 0,C 180,E1 -15165.257,E2 -15165.257} C_VEL
LIN {X 0,Y 319.55,Z 146.441,A -85,B 0,C 180,E1 -15168.763,E2 -15168.763} C_VEL
LIN {X 0,Y 322.843,Z 157.533,A -85,B 0,C 180,E1 -15172.117,E2 -15172.117} C_VEL
LIN {X 0,Y 324.308,Z 162.773,A -85,B 0,C 180,E1 -15173.556,E2 -15173.556} C_VEL
LIN {X 0,Y 332.849,Z 179.724,A -85,B 0,C 180,E1 -15175.065,E2 -15175.065} C_VEL
LIN {X 0,Y 340.548,Z 197.1,A -85,B 0,C 180,E1 -15176.39,E2 -15176.39} C_VEL
LIN {X 0,Y 343.42,Z 213.825,A -85,B 0,C 180,E1 -15177.114,E2 -15177.114} C_VEL
LIN {X 0,Y 339.748,Z 327.382,A -85,B 0,C 180,E1 -15179.506,E2 -15179.506} C_VEL
LIN {X 0,Y 338.67,Z 342.493,A -85,B 0,C 180,E1 -15180.001,E2 -15180.001} C_VEL
LIN {X 0,Y 337.053,Z 357.939,A -85,B 0,C 180,E1 -15180.744,E2 -15180.744} C_VEL
LIN {X 0,Y 335.27,Z 372.27,A -85,B 0,C 180,E1 -15181.692,E2 -15181.692} C_VEL
LIN {X 0,Y 333.17,Z 386.111,A -85,B 0,C 180,E1 -15182.86,E2 -15182.86} C_VEL
LIN {X 0,Y 330.917,Z 398.837,A -85,B 0,C 180,E1 -15184.19,E2 -15184.19} C_VEL
LIN {X 0,Y 328.456,Z 411.714,A -85,B 0,C 180,E1 -15185.844,E2 -15185.844} C_VEL
LIN {X 0,Y 326.39,Z 422.339,A -85,B 0,C 180,E1 -15187.499,E2 -15187.499} C_VEL
LIN {X 0,Y 324.438,Z 432.49,A -85,B 0,C 180,E1 -15189.39,E2 -15189.39} C_VEL
LIN {X 0,Y 322.322,Z 442.259,A -85,B 0,C 180,E1 -15191.569,E2 -15191.569} C_VEL
LIN {X 0,Y 320.739,Z 450.419,A -85,B 0,C 180,E1 -15193.777,E2 -15193.777} C_VEL
LIN {X 0,Y 319.586,Z 457.171,A -85,B 0,C 180,E1 -15196.001,E2 -15196.001} C_VEL
LIN {X 0,Y 318.591,Z 463.409,A -85,B 0,C 180,E1 -15198.548,E2 -15198.548} C_VEL
LIN {X 0,Y 318.076,Z 468.239,A -85,B 0,C 180,E1 -15201.102,E2 -15201.102} C_VEL
LIN {X 0,Y 317.808,Z 471.78,A -85,B 0,C 180,E1 -15203.652,E2 -15203.652} C_VEL
LIN {X 0,Y 317.757,Z 474.112,A -85,B 0,C 180,E1 -15206.195,E2 -15206.195} C_VEL
LIN {X 0,Y 317.738,Z 475.283,A -85,B 0,C 180,E1 -15208.733,E2 -15208.733} C_VEL
LIN {X 0,Y 317.738,Z 475.28,A -85,B 0,C 180,E1 -15211.267,E2 -15211.267} C_VEL
LIN {X 0,Y 317.758,Z 474.096,A -85,B 0,C 180,E1 -15213.804,E2 -15213.804} C_VEL
LIN {X 0,Y 317.808,Z 471.755,A -85,B 0,C 180,E1 -15216.348,E2 -15216.348} C_VEL
LIN {X 0,Y 318.076,Z 468.209,A -85,B 0,C 180,E1 -15218.898,E2 -15218.898} C_VEL
LIN {X 0,Y 318.586,Z 463.37,A -85,B 0,C 180,E1 -15221.452,E2 -15221.452} C_VEL
LIN {X 0,Y 319.568,Z 457.113,A -85,B 0,C 180,E1 -15224,E2 -15224} C_VEL
LIN {X 0,Y 320.927,Z 449.259,A -85,B 0,C 180,E1 -15226.54,E2 -15226.54} C_VEL
LIN {X 0,Y 322.533,Z 440.913,A -85,B 0,C 180,E1 -15228.748,E2 -15228.748} C_VEL
LIN {X 0,Y 324.731,Z 430.87,A -85,B 0,C 180,E1 -15230.922,E2 -15230.922} C_VEL
LIN {X 0,Y 326.713,Z 420.597,A -85,B 0,C 180,E1 -15232.781,E2 -15232.781} C_VEL
LIN {X 0,Y 329.106,Z 408.36,A -85,B 0,C 180,E1 -15234.609,E2 -15234.609} C_VEL
LIN {X 0,Y 331.398,Z 396.083,A -85,B 0,C 180,E1 -15236.107,E2 -15236.107} C_VEL
LIN {X 0,Y 333.701,Z 382.724,A -85,B 0,C 180,E1 -15237.433,E2 -15237.433} C_VEL
LIN {X 0,Y 335.715,Z 368.749,A -85,B 0,C 180,E1 -15238.546,E2 -15238.546} C_VEL
LIN {X 0,Y 337.374,Z 354.998,A -85,B 0,C 180,E1 -15239.396,E2 -15239.396} C_VEL
LIN {X 0,Y 338.816,Z 340.179,A -85,B 0,C 180,E1 -15240.071,E2 -15240.071} C_VEL
LIN {X 0,Y 339.799,Z 325.056,A -85,B 0,C 180,E1 -15240.532,E2 -15240.532} C_VEL
LIN {X 0,Y 343.332,Z 214.415,A -85,B 0,C 180,E1 -15242.856,E2 -15242.856} C_VEL
LIN {X 0,Y 340.723,Z 198.528,A -85,B 0,C 180,E1 -15243.53,E2 -15243.53} C_VEL
LIN {X 0,Y 339.725,Z 194.966,A -85,B 0,C 180,E1 -15243.729,E2 -15243.729} C_VEL
LIN {X 0,Y 330.51,Z 174.913,A -85,B 0,C 180,E1 -15245.313,E2 -15245.313} C_VEL
LIN {X 0,Y 324.173,Z 162.394,A -85,B 0,C 180,E1 -15246.458,E2 -15246.458} C_VEL
LIN {X 0,Y 320.807,Z 150.514,A -85,B 0,C 180,E1 -15249.937,E2 -15249.937} C_VEL
LIN {X 0,Y 319.529,Z 146.307,A -85,B 0,C 180,E1 -15251.288,E2 -15251.288} C_VEL
LIN {X 0,Y 319.489,Z 146.309,A -85,B 0,C 180,E1 -15254.743,E2 -15254.743} C_VEL
LIN {X 0,Y 319.526,Z 146.306,A -85,B 0,C 180,E1 -15258.403,E2 -15258.403} C_VEL
LIN {X 0,Y 319.544,Z 146.301,A -85,B 0,C 180,E1 -15261.988,E2 -15261.988} C_VEL
LIN {X 0,Y 319.561,Z 146.299,A -85,B 0,C 180,E1 -15265.124,E2 -15265.124} C_VEL
LIN {X 0,Y 319.571,Z 146.3,A -85,B 0,C 180,E1 -15269.058,E2 -15269.058} C_VEL
LIN {X 0,Y 319.61,Z 146.295,A -85,B 0,C 180,E1 -15272.498,E2 -15272.498} C_VEL
LIN {X 0,Y 319.605,Z 146.297,A -85,B 0,C 180,E1 -15275.304,E2 -15275.304} C_VEL
LIN {X 0,Y 319.598,Z 146.299,A -85,B 0,C 180,E1 -15278.048,E2 -15278.048} C_VEL
LIN {X 0,Y 319.69,Z 146.285,A -85,B 0,C 180,E1 -15280.963,E2 -15280.963} C_VEL
LIN {X 0,Y 319.733,Z 146.283,A -85,B 0,C 180,E1 -15285.276,E2 -15285.276} C_VEL
LIN {X 0,Y 319.717,Z 146.28,A -85,B 0,C 180,E1 -15288.59,E2 -15288.59} C_VEL
LIN {X 0,Y 319.855,Z 146.26,A -85,B 0,C 180,E1 -15292.425,E2 -15292.425} C_VEL
LIN {X 0,Y 319.73,Z 146.278,A -85,B 0,C 180,E1 -15294.956,E2 -15294.956} C_VEL
LIN {X 0,Y 319.986,Z 146.249,A -85,B 0,C 180,E1 -15297.483,E2 -15297.483} C_VEL
LIN {X 0,Y 320.015,Z 146.244,A -85,B 0,C 180,E1 -15301.259,E2 -15301.259} C_VEL
LIN {X 0,Y 319.723,Z 146.277,A -85,B 0,C 180,E1 -15305.044,E2 -15305.044} C_VEL
LIN {X 0,Y 319.855,Z 146.267,A -85,B 0,C 180,E1 -15307.576,E2 -15307.576} C_VEL
LIN {X 0,Y 319.716,Z 146.285,A -85,B 0,C 180,E1 -15311.411,E2 -15311.411} C_VEL
LIN {X 0,Y 319.666,Z 146.291,A -85,B 0,C 180,E1 -15314.678,E2 -15314.678} C_VEL
LIN {X 0,Y 319.659,Z 146.291,A -85,B 0,C 180,E1 -15319.021,E2 -15319.021} C_VEL
LIN {X 0,Y 319.553,Z 146.306,A -85,B 0,C 180,E1 -15323.321,E2 -15323.321} C_VEL
LIN {X 0,Y 319.568,Z 146.274,A -85,B 0,C 180,E1 -15326.094,E2 -15326.094} C_VEL
LIN {X 0,Y 319.542,Z 146.303,A -85,B 0,C 180,E1 -15328.938,E2 -15328.938} C_VEL
LIN {X 0,Y 319.525,Z 146.306,A -85,B 0,C 180,E1 -15331.863,E2 -15331.863} C_VEL
LIN {X 0,Y 319.581,Z 146.302,A -85,B 0,C 180,E1 -15335.543,E2 -15335.543} C_VEL
LIN {X 0,Y 319.529,Z 146.302,A -85,B 0,C 180,E1 -15339.662,E2 -15339.662} C_VEL
LIN {X 0,Y 319.519,Z 146.309,A -85,B 0,C 180,E1 -15343.46,E2 -15343.46} C_VEL
LIN {X 0,Y 319.551,Z 146.304,A -85,B 0,C 180,E1 -15347.016,E2 -15347.016} C_VEL
LIN {X 0,Y 319.515,Z 146.306,A -85,B 0,C 180,E1 -15350.366,E2 -15350.366} C_VEL
LIN {X 0,Y 319.577,Z 146.405,A -85,B 0,C 180,E1 -15352.428,E2 -15352.428} C_VEL
LIN {X 0,Y 320.234,Z 148.516,A -85,B 0,C 180,E1 -15353.1,E2 -15353.1} C_VEL
LIN {X 0,Y 329.737,Z 165.837,A -85,B 0,C 180,E1 -15354.794,E2 -15354.794} C_VEL
LIN {X 0,Y 337.125,Z 180.544,A -85,B 0,C 180,E1 -15356.054,E2 -15356.054} C_VEL
LIN {X 0,Y 343.785,Z 195.512,A -85,B 0,C 180,E1 -15357.171,E2 -15357.171} C_VEL
LIN {X 0,Y 341.221,Z 277.023,A -85,B 0,C 180,E1 -15358.879,E2 -15358.879} C_VEL
LIN {X 0,Y 339.91,Z 314.185,A -85,B 0,C 180,E1 -15359.693,E2 -15359.693} C_VEL
LIN {X 0,Y 338.938,Z 328.92,A -85,B 0,C 180,E1 -15360.234,E2 -15360.234} C_VEL
LIN {X 0,Y 337.559,Z 343.828,A -85,B 0,C 180,E1 -15361.021,E2 -15361.021} C_VEL
LIN {X 0,Y 335.767,Z 358.728,A -85,B 0,C 180,E1 -15362.074,E2 -15362.074} C_VEL
LIN {X 0,Y 333.793,Z 371.974,A -85,B 0,C 180,E1 -15363.253,E2 -15363.253} C_VEL
LIN {X 0,Y 331.473,Z 385.433,A -85,B 0,C 180,E1 -15364.742,E2 -15364.742} C_VEL
LIN {X 0,Y 329.172,Z 397.601,A -85,B 0,C 180,E1 -15366.395,E2 -15366.395} C_VEL
LIN {X 0,Y 327.006,Z 408.758,A -85,B 0,C 180,E1 -15368.239,E2 -15368.239} C_VEL
LIN {X 0,Y 324.992,Z 418.107,A -85,B 0,C 180,E1 -15370.087,E2 -15370.087} C_VEL
LIN {X 0,Y 322.999,Z 427.298,A -85,B 0,C 180,E1 -15372.265,E2 -15372.265} C_VEL
LIN {X 0,Y 321.171,Z 435.935,A -85,B 0,C 180,E1 -15374.776,E2 -15374.776} C_VEL
LIN {X 0,Y 320.226,Z 441.266,A -85,B 0,C 180,E1 -15376.677,E2 -15376.677} C_VEL
LIN {X 0,Y 319.161,Z 447.081,A -85,B 0,C 180,E1 -15379.212,E2 -15379.212} C_VEL
LIN {X 0,Y 318.641,Z 450.521,A -85,B 0,C 180,E1 -15381.118,E2 -15381.118} C_VEL
LIN {X 0,Y 318.16,Z 454.093,A -85,B 0,C 180,E1 -15383.736,E2 -15383.736} C_VEL
LIN {X 0,Y 317.938,Z 456.308,A -85,B 0,C 180,E1 -15386.198,E2 -15386.198} C_VEL
LIN {X 0,Y 317.778,Z 457.485,A -85,B 0,C 180,E1 -15388.733,E2 -15388.733} C_VEL
LIN {X 0,Y 317.778,Z 457.499,A -85,B 0,C 180,E1 -15391.267,E2 -15391.267} C_VEL
LIN {X 0,Y 317.937,Z 456.38,A -85,B 0,C 180,E1 -15393.802,E2 -15393.802} C_VEL
LIN {X 0,Y 318.174,Z 454.134,A -85,B 0,C 180,E1 -15396.341,E2 -15396.341} C_VEL
LIN {X 0,Y 318.612,Z 450.702,A -85,B 0,C 180,E1 -15398.883,E2 -15398.883} C_VEL
LIN {X 0,Y 319.341,Z 446.001,A -85,B 0,C 180,E1 -15401.424,E2 -15401.424} C_VEL
LIN {X 0,Y 320.543,Z 439.904,A -85,B 0,C 180,E1 -15403.956,E2 -15403.956} C_VEL
LIN {X 0,Y 321.983,Z 432.229,A -85,B 0,C 180,E1 -15406.485,E2 -15406.485} C_VEL
LIN {X 0,Y 323.725,Z 424.039,A -85,B 0,C 180,E1 -15408.676,E2 -15408.676} C_VEL
LIN {X 0,Y 325.825,Z 414.168,A -85,B 0,C 180,E1 -15410.849,E2 -15410.849} C_VEL
LIN {X 0,Y 327.933,Z 404.045,A -85,B 0,C 180,E1 -15412.691,E2 -15412.691} C_VEL
LIN {X 0,Y 330.24,Z 391.989,A -85,B 0,C 180,E1 -15414.519,E2 -15414.519} C_VEL
LIN {X 0,Y 332.476,Z 379.893,A -85,B 0,C 180,E1 -15416.016,E2 -15416.016} C_VEL
LIN {X 0,Y 334.655,Z 366.745,A -85,B 0,C 180,E1 -15417.348,E2 -15417.348} C_VEL
LIN {X 0,Y 336.368,Z 354.213,A -85,B 0,C 180,E1 -15418.381,E2 -15418.381} C_VEL
LIN {X 0,Y 337.922,Z 340.447,A -85,B 0,C 180,E1 -15419.284,E2 -15419.284} C_VEL
LIN {X 0,Y 339.201,Z 326.102,A -85,B 0,C 180,E1 -15419.991,E2 -15419.991} C_VEL
LIN {X 0,Y 340.211,Z 311.051,A -85,B 0,C 180,E1 -15420.491,E2 -15420.491} C_VEL
LIN {X 0,Y 341.296,Z 276.585,A -85,B 0,C 180,E1 -15421.238,E2 -15421.238} C_VEL
LIN {X 0,Y 340.94,Z 270.78,A -85,B 0,C 180,E1 -15421.415,E2 -15421.415} C_VEL
LIN {X 0,Y 336.72,Z 252.128,A -85,B 0,C 180,E1 -15422.318,E2 -15422.318} C_VEL
LIN {X 0,Y 336.33,Z 246.325,A -85,B 0,C 180,E1 -15422.505,E2 -15422.505} C_VEL
LIN {X 0,Y 337.879,Z 197.666,A -85,B 0,C 180,E1 -15423.546,E2 -15423.546} C_VEL
LIN {X 0,Y 330.303,Z 180.859,A -85,B 0,C 180,E1 -15424.864,E2 -15424.864} C_VEL
LIN {X 0,Y 321.611,Z 163.958,A -85,B 0,C 180,E1 -15426.416,E2 -15426.416} C_VEL
LIN {X 0,Y 314.728,Z 152.009,A -85,B 0,C 180,E1 -15427.689,E2 -15427.689} C_VEL
LIN {X 0,Y 312.826,Z 148.599,A -85,B 0,C 180,E1 -15428.077,E2 -15428.077} C_VEL
LIN {X 0,Y 312.446,Z 147.189,A -85,B 0,C 180,E1 -15428.636,E2 -15428.636} C_VEL
LIN {X 0,Y 312.465,Z 147.187,A -85,B 0,C 180,E1 -15432.436,E2 -15432.436} C_VEL
LIN {X 0,Y 312.457,Z 147.186,A -85,B 0,C 180,E1 -15436.035,E2 -15436.035} C_VEL
LIN {X 0,Y 312.456,Z 147.189,A -85,B 0,C 180,E1 -15439.886,E2 -15439.886} C_VEL
LIN {X 0,Y 312.534,Z 147.168,A -85,B 0,C 180,E1 -15444.051,E2 -15444.051} C_VEL
LIN {X 0,Y 312.501,Z 147.167,A -85,B 0,C 180,E1 -15447.333,E2 -15447.333} C_VEL
LIN {X 0,Y 312.499,Z 147.182,A -85,B 0,C 180,E1 -15451.295,E2 -15451.295} C_VEL
LIN {X 0,Y 312.522,Z 147.177,A -85,B 0,C 180,E1 -15454.705,E2 -15454.705} C_VEL
LIN {X 0,Y 312.541,Z 147.171,A -85,B 0,C 180,E1 -15457.525,E2 -15457.525} C_VEL
LIN {X 0,Y 312.553,Z 147.169,A -85,B 0,C 180,E1 -15461.651,E2 -15461.651} C_VEL
LIN {X 0,Y 312.685,Z 147.154,A -85,B 0,C 180,E1 -15465.686,E2 -15465.686} C_VEL
LIN {X 0,Y 312.688,Z 147.156,A -85,B 0,C 180,E1 -15469.641,E2 -15469.641} C_VEL
LIN {X 0,Y 312.798,Z 147.146,A -85,B 0,C 180,E1 -15472.252,E2 -15472.252} C_VEL
LIN {X 0,Y 312.689,Z 147.152,A -85,B 0,C 180,E1 -15474.842,E2 -15474.842} C_VEL
LIN {X 0,Y 312.981,Z 147.121,A -85,B 0,C 180,E1 -15478.713,E2 -15478.713} C_VEL
LIN {X 0,Y 312.932,Z 147.129,A -85,B 0,C 180,E1 -15482.574,E2 -15482.574} C_VEL
LIN {X 0,Y 312.845,Z 147.14,A -85,B 0,C 180,E1 -15486.449,E2 -15486.449} C_VEL
LIN {X 0,Y 312.753,Z 147.144,A -85,B 0,C 180,E1 -15489.05,E2 -15489.05} C_VEL
LIN {X 0,Y 312.637,Z 147.162,A -85,B 0,C 180,E1 -15492.991,E2 -15492.991} C_VEL
LIN {X 0,Y 312.624,Z 147.172,A -85,B 0,C 180,E1 -15495.65,E2 -15495.65} C_VEL
LIN {X 0,Y 312.566,Z 147.178,A -85,B 0,C 180,E1 -15499.711,E2 -15499.711} C_VEL
LIN {X 0,Y 312.528,Z 147.174,A -85,B 0,C 180,E1 -15502.78,E2 -15502.78} C_VEL
LIN {X 0,Y 312.539,Z 147.173,A -85,B 0,C 180,E1 -15505.911,E2 -15505.911} C_VEL
LIN {X 0,Y 312.505,Z 147.183,A -85,B 0,C 180,E1 -15509.654,E2 -15509.654} C_VEL
LIN {X 0,Y 312.521,Z 147.172,A -85,B 0,C 180,E1 -15513.689,E2 -15513.689} C_VEL
LIN {X 0,Y 312.527,Z 147.174,A -85,B 0,C 180,E1 -15517.385,E2 -15517.385} C_VEL
LIN {X 0,Y 312.491,Z 147.183,A -85,B 0,C 180,E1 -15520.709,E2 -15520.709} C_VEL
LIN {X 0,Y 312.452,Z 147.189,A -85,B 0,C 180,E1 -15524.209,E2 -15524.209} C_VEL
LIN {X 0,Y 312.501,Z 147.261,A -85,B 0,C 180,E1 -15527.915,E2 -15527.915} C_VEL
LIN {X 0,Y 315.863,Z 158.584,A -85,B 0,C 180,E1 -15531.464,E2 -15531.464} C_VEL
LIN {X 0,Y 316.964,Z 162.434,A -85,B 0,C 180,E1 -15532.566,E2 -15532.566} C_VEL
LIN {X 0,Y 325.803,Z 179.61,A -85,B 0,C 180,E1 -15534.197,E2 -15534.197} C_VEL
LIN {X 0,Y 334.481,Z 198.778,A -85,B 0,C 180,E1 -15535.744,E2 -15535.744} C_VEL
LIN {X 0,Y 335.43,Z 202.873,A -85,B 0,C 180,E1 -15535.957,E2 -15535.957} C_VEL
LIN {X 0,Y 337.436,Z 215.612,A -85,B 0,C 180,E1 -15536.504,E2 -15536.504} C_VEL
LIN {X 0,Y 333.585,Z 328.704,A -85,B 0,C 180,E1 -15538.924,E2 -15538.924} C_VEL
LIN {X 0,Y 332.394,Z 344.136,A -85,B 0,C 180,E1 -15539.462,E2 -15539.462} C_VEL
LIN {X 0,Y 330.713,Z 359.049,A -85,B 0,C 180,E1 -15540.215,E2 -15540.215} C_VEL
LIN {X 0,Y 328.905,Z 372.994,A -85,B 0,C 180,E1 -15541.173,E2 -15541.173} C_VEL
LIN {X 0,Y 326.846,Z 385.917,A -85,B 0,C 180,E1 -15542.29,E2 -15542.29} C_VEL
LIN {X 0,Y 324.483,Z 398.64,A -85,B 0,C 180,E1 -15543.64,E2 -15543.64} C_VEL
LIN {X 0,Y 321.911,Z 411.516,A -85,B 0,C 180,E1 -15545.32,E2 -15545.32} C_VEL
LIN {X 0,Y 319.746,Z 422.305,A -85,B 0,C 180,E1 -15547.037,E2 -15547.037} C_VEL
LIN {X 0,Y 317.749,Z 432.291,A -85,B 0,C 180,E1 -15548.935,E2 -15548.935} C_VEL
LIN {X 0,Y 315.51,Z 442.06,A -85,B 0,C 180,E1 -15551.156,E2 -15551.156} C_VEL
LIN {X 0,Y 313.843,Z 450.219,A -85,B 0,C 180,E1 -15553.41,E2 -15553.41} C_VEL
LIN {X 0,Y 312.631,Z 456.972,A -85,B 0,C 180,E1 -15555.683,E2 -15555.683} C_VEL
LIN {X 0,Y 311.594,Z 463.21,A -85,B 0,C 180,E1 -15558.288,E2 -15558.288} C_VEL
LIN {X 0,Y 311.001,Z 468.039,A -85,B 0,C 180,E1 -15560.898,E2 -15560.898} C_VEL
LIN {X 0,Y 310.713,Z 471.581,A -85,B 0,C 180,E1 -15563.506,E2 -15563.506} C_VEL
LIN {X 0,Y 310.67,Z 473.913,A -85,B 0,C 180,E1 -15566.108,E2 -15566.108} C_VEL
LIN {X 0,Y 310.652,Z 475.084,A -85,B 0,C 180,E1 -15568.704,E2 -15568.704} C_VEL
LIN {X 0,Y 310.652,Z 475.081,A -85,B 0,C 180,E1 -15571.296,E2 -15571.296} C_VEL
LIN {X 0,Y 310.671,Z 473.897,A -85,B 0,C 180,E1 -15573.891,E2 -15573.891} C_VEL
LIN {X 0,Y 310.713,Z 471.554,A -85,B 0,C 180,E1 -15576.494,E2 -15576.494} C_VEL
LIN {X 0,Y 311,Z 468.008,A -85,B 0,C 180,E1 -15579.102,E2 -15579.102} C_VEL
LIN {X 0,Y 311.589,Z 463.169,A -85,B 0,C 180,E1 -15581.712,E2 -15581.712} C_VEL
LIN {X 0,Y 312.604,Z 456.91,A -85,B 0,C 180,E1 -15584.318,E2 -15584.318} C_VEL
LIN {X 0,Y 314.055,Z 449.057,A -85,B 0,C 180,E1 -15586.913,E2 -15586.913} C_VEL
LIN {X 0,Y 315.726,Z 440.71,A -85,B 0,C 180,E1 -15589.168,E2 -15589.168} C_VEL
LIN {X 0,Y 318.027,Z 430.666,A -85,B 0,C 180,E1 -15591.385,E2 -15591.385} C_VEL
LIN {X 0,Y 320.11,Z 420.393,A -85,B 0,C 180,E1 -15593.278,E2 -15593.278} C_VEL
LIN {X 0,Y 322.629,Z 408.157,A -85,B 0,C 180,E1 -15595.137,E2 -15595.137} C_VEL
LIN {X 0,Y 325.256,Z 394.535,A -85,B 0,C 180,E1 -15596.812,E2 -15596.812} C_VEL
LIN {X 0,Y 327.666,Z 380.881,A -85,B 0,C 180,E1 -15598.156,E2 -15598.156} C_VEL
LIN {X 0,Y 329.657,Z 367.325,A -85,B 0,C 180,E1 -15599.227,E2 -15599.227} C_VEL
LIN {X 0,Y 331.51,Z 352.167,A -85,B 0,C 180,E1 -15600.144,E2 -15600.144} C_VEL
LIN {X 0,Y 332.926,Z 337.213,A -85,B 0,C 180,E1 -15600.791,E2 -15600.791} C_VEL
LIN {X 0,Y 333.867,Z 321.826,A -85,B 0,C 180,E1 -15601.223,E2 -15601.223} C_VEL
LIN {X 0,Y 337.312,Z 214.438,A -85,B 0,C 180,E1 -15603.513,E2 -15603.513} C_VEL
LIN {X 0,Y 334.532,Z 198.821,A -85,B 0,C 180,E1 -15604.222,E2 -15604.222} C_VEL
LIN {X 0,Y 325.283,Z 178.56,A -85,B 0,C 180,E1 -15605.866,E2 -15605.866} C_VEL
LIN {X 0,Y 318.612,Z 165.697,A -85,B 0,C 180,E1 -15607.085,E2 -15607.085} C_VEL
LIN {X 0,Y 316.841,Z 162.039,A -85,B 0,C 180,E1 -15607.47,E2 -15607.47} C_VEL
LIN {X 0,Y 313.553,Z 150.807,A -85,B 0,C 180,E1 -15610.908,E2 -15610.908} C_VEL
LIN {X 0,Y 312.484,Z 147.185,A -85,B 0,C 180,E1 -15612.082,E2 -15612.082} C_VEL
LIN {X 0,Y 312.459,Z 147.188,A -85,B 0,C 180,E1 -15616.035,E2 -15616.035} C_VEL
LIN {X 0,Y 312.504,Z 147.181,A -85,B 0,C 180,E1 -15619.875,E2 -15619.875} C_VEL
LIN {X 0,Y 312.536,Z 147.171,A -85,B 0,C 180,E1 -15624.051,E2 -15624.051} C_VEL
LIN {X 0,Y 312.505,Z 147.176,A -85,B 0,C 180,E1 -15627.334,E2 -15627.334} C_VEL
LIN {X 0,Y 312.553,Z 147.176,A -85,B 0,C 180,E1 -15631.276,E2 -15631.276} C_VEL
LIN {X 0,Y 312.586,Z 147.173,A -85,B 0,C 180,E1 -15634.711,E2 -15634.711} C_VEL
LIN {X 0,Y 312.588,Z 147.173,A -85,B 0,C 180,E1 -15637.529,E2 -15637.529} C_VEL
LIN {X 0,Y 312.64,Z 147.166,A -85,B 0,C 180,E1 -15641.657,E2 -15641.657} C_VEL
LIN {X 0,Y 312.696,Z 147.159,A -85,B 0,C 180,E1 -15645.686,E2 -15645.686} C_VEL
LIN {X 0,Y 312.687,Z 147.16,A -85,B 0,C 180,E1 -15649.642,E2 -15649.642} C_VEL
LIN {X 0,Y 312.798,Z 147.138,A -85,B 0,C 180,E1 -15652.253,E2 -15652.253} C_VEL
LIN {X 0,Y 312.699,Z 147.154,A -85,B 0,C 180,E1 -15654.842,E2 -15654.842} C_VEL
LIN {X 0,Y 312.932,Z 147.128,A -85,B 0,C 180,E1 -15657.426,E2 -15657.426} C_VEL
LIN {X 0,Y 312.982,Z 147.12,A -85,B 0,C 180,E1 -15661.287,E2 -15661.287} C_VEL
LIN {X 0,Y 312.844,Z 147.143,A -85,B 0,C 180,E1 -15666.449,E2 -15666.449} C_VEL
LIN {X 0,Y 312.752,Z 147.142,A -85,B 0,C 180,E1 -15669.05,E2 -15669.05} C_VEL
LIN {X 0,Y 312.626,Z 147.158,A -85,B 0,C 180,E1 -15672.992,E2 -15672.992} C_VEL
LIN {X 0,Y 312.576,Z 147.176,A -85,B 0,C 180,E1 -15675.653,E2 -15675.653} C_VEL
LIN {X 0,Y 312.565,Z 147.176,A -85,B 0,C 180,E1 -15679.711,E2 -15679.711} C_VEL
LIN {X 0,Y 312.523,Z 147.18,A -85,B 0,C 180,E1 -15682.779,E2 -15682.779} C_VEL
LIN {X 0,Y 312.529,Z 147.152,A -85,B 0,C 180,E1 -15685.907,E2 -15685.907} C_VEL
LIN {X 0,Y 312.496,Z 147.186,A -85,B 0,C 180,E1 -15689.655,E2 -15689.655} C_VEL
LIN {X 0,Y 312.521,Z 147.177,A -85,B 0,C 180,E1 -15693.689,E2 -15693.689} C_VEL
LIN {X 0,Y 312.515,Z 147.176,A -85,B 0,C 180,E1 -15697.387,E2 -15697.387} C_VEL
LIN {X 0,Y 312.441,Z 147.187,A -85,B 0,C 180,E1 -15700.717,E2 -15700.717} C_VEL
LIN {X 0,Y 312.451,Z 147.186,A -85,B 0,C 180,E1 -15704.21,E2 -15704.21} C_VEL
LIN {X 0,Y 312.455,Z 147.191,A -85,B 0,C 180,E1 -15707.925,E2 -15707.925} C_VEL
LIN {X 0,Y 312.507,Z 147.37,A -85,B 0,C 180,E1 -15711.638,E2 -15711.638} C_VEL
LIN {X 0,Y 312.916,Z 148.884,A -85,B 0,C 180,E1 -15712.089,E2 -15712.089} C_VEL
LIN {X 0,Y 320.505,Z 161.97,A -85,B 0,C 180,E1 -15713.506,E2 -15713.506} C_VEL
LIN {X 0,Y 329.371,Z 178.9,A -85,B 0,C 180,E1 -15715.091,E2 -15715.091} C_VEL
LIN {X 0,Y 337.353,Z 196.504,A -85,B 0,C 180,E1 -15716.482,E2 -15716.482} C_VEL
LIN {X 0,Y 337.838,Z 198.391,A -85,B 0,C 180,E1 -15716.584,E2 -15716.584} C_VEL
LIN {X 0,Y 333.899,Z 313.239,A -85,B 0,C 180,E1 -15719.045,E2 -15719.045} C_VEL
LIN {X 0,Y 332.924,Z 327.562,A -85,B 0,C 180,E1 -15719.56,E2 -15719.56} C_VEL
LIN {X 0,Y 331.626,Z 341.626,A -85,B 0,C 180,E1 -15720.285,E2 -15720.285} C_VEL
LIN {X 0,Y 330.017,Z 355.075,A -85,B 0,C 180,E1 -15721.196,E2 -15721.196} C_VEL
LIN {X 0,Y 327.977,Z 369.044,A -85,B 0,C 180,E1 -15722.394,E2 -15722.394} C_VEL
LIN {X 0,Y 325.769,Z 381.814,A -85,B 0,C 180,E1 -15723.752,E2 -15723.752} C_VEL
LIN {X 0,Y 323.25,Z 394.677,A -85,B 0,C 180,E1 -15725.43,E2 -15725.43} C_VEL
LIN {X 0,Y 321.423,Z 403.65,A -85,B 0,C 180,E1 -15726.823,E2 -15726.823} C_VEL
LIN {X 0,Y 319.238,Z 413.832,A -85,B 0,C 180,E1 -15728.7,E2 -15728.7} C_VEL
LIN {X 0,Y 317.084,Z 423.79,A -85,B 0,C 180,E1 -15730.918,E2 -15730.918} C_VEL
LIN {X 0,Y 315.148,Z 432.049,A -85,B 0,C 180,E1 -15733.148,E2 -15733.148} C_VEL
LIN {X 0,Y 313.645,Z 439.796,A -85,B 0,C 180,E1 -15735.731,E2 -15735.731} C_VEL
LIN {X 0,Y 312.38,Z 445.964,A -85,B 0,C 180,E1 -15738.318,E2 -15738.318} C_VEL
LIN {X 0,Y 311.601,Z 450.722,A -85,B 0,C 180,E1 -15740.916,E2 -15740.916} C_VEL
LIN {X 0,Y 311.057,Z 454.512,A -85,B 0,C 180,E1 -15743.792,E2 -15743.792} C_VEL
LIN {X 0,Y 310.873,Z 456.507,A -85,B 0,C 180,E1 -15746.111,E2 -15746.111} C_VEL
LIN {X 0,Y 310.691,Z 457.683,A -85,B 0,C 180,E1 -15748.704,E2 -15748.704} C_VEL
LIN {X 0,Y 310.691,Z 457.697,A -85,B 0,C 180,E1 -15751.296,E2 -15751.296} C_VEL
LIN {X 0,Y 310.872,Z 456.578,A -85,B 0,C 180,E1 -15753.889,E2 -15753.889} C_VEL
LIN {X 0,Y 311.109,Z 454.332,A -85,B 0,C 180,E1 -15756.486,E2 -15756.486} C_VEL
LIN {X 0,Y 311.575,Z 450.9,A -85,B 0,C 180,E1 -15759.085,E2 -15759.085} C_VEL
LIN {X 0,Y 312.352,Z 446.2,A -85,B 0,C 180,E1 -15761.683,E2 -15761.683} C_VEL
LIN {X 0,Y 313.616,Z 440.102,A -85,B 0,C 180,E1 -15764.271,E2 -15764.271} C_VEL
LIN {X 0,Y 315.128,Z 432.427,A -85,B 0,C 180,E1 -15766.854,E2 -15766.854} C_VEL
LIN {X 0,Y 316.968,Z 424.236,A -85,B 0,C 180,E1 -15769.09,E2 -15769.09} C_VEL
LIN {X 0,Y 319.17,Z 414.365,A -85,B 0,C 180,E1 -15771.305,E2 -15771.305} C_VEL
LIN {X 0,Y 321.342,Z 404.242,A -85,B 0,C 180,E1 -15773.183,E2 -15773.183} C_VEL
LIN {X 0,Y 323.798,Z 392.184,A -85,B 0,C 180,E1 -15775.04,E2 -15775.04} C_VEL
LIN {X 0,Y 326.096,Z 380.088,A -85,B 0,C 180,E1 -15776.565,E2 -15776.565} C_VEL
LIN {X 0,Y 328.364,Z 366.938,A -85,B 0,C 180,E1 -15777.917,E2 -15777.917} C_VEL
LIN {X 0,Y 330.279,Z 353.182,A -85,B 0,C 180,E1 -15779.061,E2 -15779.061} C_VEL
LIN {X 0,Y 331.908,Z 339.209,A -85,B 0,C 180,E1 -15779.964,E2 -15779.964} C_VEL
LIN {X 0,Y 333.209,Z 324.461,A -85,B 0,C 180,E1 -15780.675,E2 -15780.675} C_VEL
LIN {X 0,Y 334.146,Z 309.727,A -85,B 0,C 180,E1 -15781.15,E2 -15781.15} C_VEL
LIN {X 0,Y 336.33,Z 246.325,A -85,B 0,C 180,E1 -15782.505,E2 -15782.505} C_VEL
LIN {X 0,Y 335.935,Z 240.528,A -85,B 0,C 180,E1 -15782.693,E2 -15782.693} C_VEL
LIN {X 0,Y 331.755,Z 221.922,A -85,B 0,C 180,E1 -15783.634,E2 -15783.634} C_VEL
LIN {X 0,Y 331.427,Z 216.124,A -85,B 0,C 180,E1 -15783.82,E2 -15783.82} C_VEL
LIN {X 0,Y 331.914,Z 199.731,A -85,B 0,C 180,E1 -15784.183,E2 -15784.183} C_VEL
LIN {X 0,Y 324.297,Z 182.825,A -85,B 0,C 180,E1 -15785.559,E2 -15785.559} C_VEL
LIN {X 0,Y 314.969,Z 164.9,A -85,B 0,C 180,E1 -15787.292,E2 -15787.292} C_VEL
LIN {X 0,Y 307.487,Z 152.252,A -85,B 0,C 180,E1 -15788.739,E2 -15788.739} C_VEL
LIN {X 0,Y 305.868,Z 149.79,A -85,B 0,C 180,E1 -15789.057,E2 -15789.057} C_VEL
LIN {X 0,Y 305.54,Z 148.714,A -85,B 0,C 180,E1 -15789.196,E2 -15789.196} C_VEL
LIN {X 0,Y 305.409,Z 148.058,A -85,B 0,C 180,E1 -15789.479,E2 -15789.479} C_VEL
LIN {X 0,Y 305.421,Z 148.066,A -85,B 0,C 180,E1 -15793.656,E2 -15793.656} C_VEL
LIN {X 0,Y 305.435,Z 148.045,A -85,B 0,C 180,E1 -15797.419,E2 -15797.419} C_VEL
LIN {X 0,Y 305.449,Z 148.046,A -85,B 0,C 180,E1 -15801.593,E2 -15801.593} C_VEL
LIN {X 0,Y 305.462,Z 148.058,A -85,B 0,C 180,E1 -15804.887,E2 -15804.887} C_VEL
LIN {X 0,Y 305.44,Z 148.035,A -85,B 0,C 180,E1 -15808.359,E2 -15808.359} C_VEL
LIN {X 0,Y 305.465,Z 148.055,A -85,B 0,C 180,E1 -15811.108,E2 -15811.108} C_VEL
LIN {X 0,Y 305.48,Z 148.051,A -85,B 0,C 180,E1 -15814.079,E2 -15814.079} C_VEL
LIN {X 0,Y 305.461,Z 148.054,A -85,B 0,C 180,E1 -15818.4,E2 -15818.4} C_VEL
LIN {X 0,Y 305.511,Z 148.049,A -85,B 0,C 180,E1 -15821.212,E2 -15821.212} C_VEL
LIN {X 0,Y 305.626,Z 148.035,A -85,B 0,C 180,E1 -15825.348,E2 -15825.348} C_VEL
LIN {X 0,Y 305.627,Z 148.039,A -85,B 0,C 180,E1 -15829.399,E2 -15829.399} C_VEL
LIN {X 0,Y 305.748,Z 148.021,A -85,B 0,C 180,E1 -15832.072,E2 -15832.072} C_VEL
LIN {X 0,Y 305.66,Z 148.028,A -85,B 0,C 180,E1 -15834.723,E2 -15834.723} C_VEL
LIN {X 0,Y 305.948,Z 147.997,A -85,B 0,C 180,E1 -15838.684,E2 -15838.684} C_VEL
LIN {X 0,Y 305.942,Z 147.995,A -85,B 0,C 180,E1 -15841.316,E2 -15841.316} C_VEL
LIN {X 0,Y 305.668,Z 148.025,A -85,B 0,C 180,E1 -15845.277,E2 -15845.277} C_VEL
LIN {X 0,Y 305.749,Z 148.022,A -85,B 0,C 180,E1 -15847.927,E2 -15847.927} C_VEL
LIN {X 0,Y 305.602,Z 148.044,A -85,B 0,C 180,E1 -15851.945,E2 -15851.945} C_VEL
LIN {X 0,Y 305.611,Z 148.039,A -85,B 0,C 180,E1 -15855.014,E2 -15855.014} C_VEL
LIN {X 0,Y 305.548,Z 148.049,A -85,B 0,C 180,E1 -15859.429,E2 -15859.429} C_VEL
LIN {X 0,Y 305.488,Z 148.052,A -85,B 0,C 180,E1 -15863.039,E2 -15863.039} C_VEL
LIN {X 0,Y 305.479,Z 148.051,A -85,B 0,C 180,E1 -15866.2,E2 -15866.2} C_VEL
LIN {X 0,Y 305.464,Z 148.06,A -85,B 0,C 180,E1 -15869.038,E2 -15869.038} C_VEL
LIN {X 0,Y 305.439,Z 148.064,A -85,B 0,C 180,E1 -15871.953,E2 -15871.953} C_VEL
LIN {X 0,Y 305.464,Z 148.061,A -85,B 0,C 180,E1 -15875.113,E2 -15875.113} C_VEL
LIN {X 0,Y 305.45,Z 148.064,A -85,B 0,C 180,E1 -15878.529,E2 -15878.529} C_VEL
LIN {X 0,Y 305.456,Z 148.057,A -85,B 0,C 180,E1 -15882.586,E2 -15882.586} C_VEL
LIN {X 0,Y 305.43,Z 148.184,A -85,B 0,C 180,E1 -15887.044,E2 -15887.044} C_VEL
LIN {X 0,Y 308.854,Z 159.312,A -85,B 0,C 180,E1 -15890.685,E2 -15890.685} C_VEL
LIN {X 0,Y 309.632,Z 162.156,A -85,B 0,C 180,E1 -15891.519,E2 -15891.519} C_VEL
LIN {X 0,Y 318.874,Z 179.699,A -85,B 0,C 180,E1 -15893.303,E2 -15893.303} C_VEL
LIN {X 0,Y 327.49,Z 198.374,A -85,B 0,C 180,E1 -15894.902,E2 -15894.902} C_VEL
LIN {X 0,Y 329.327,Z 203.054,A -85,B 0,C 180,E1 -15895.246,E2 -15895.246} C_VEL
LIN {X 0,Y 331.45,Z 215.846,A -85,B 0,C 180,E1 -15895.827,E2 -15895.827} C_VEL
LIN {X 0,Y 328.363,Z 306.603,A -85,B 0,C 180,E1 -15897.786,E2 -15897.786} C_VEL
LIN {X 0,Y 327.39,Z 330.904,A -85,B 0,C 180,E1 -15898.359,E2 -15898.359} C_VEL
LIN {X 0,Y 326.133,Z 345.546,A -85,B 0,C 180,E1 -15898.901,E2 -15898.901} C_VEL
